KUKA KRL program: filwin67start.src

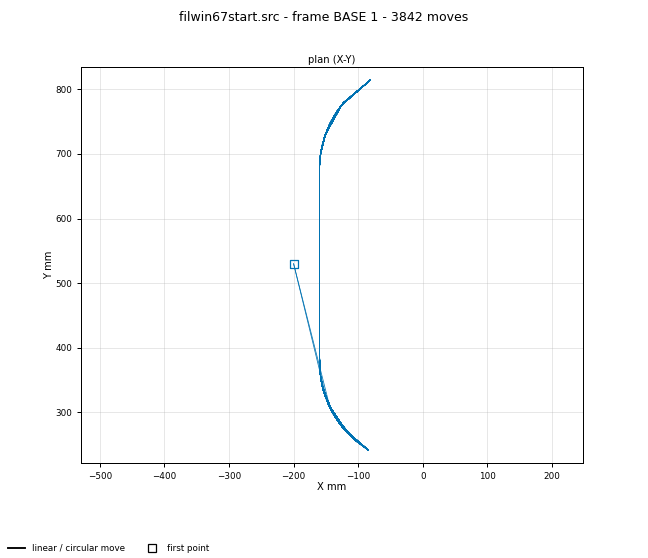
[picture p0: tool path of filwin67start.src in frame BASE 1, 3842 of 3843 moves have a stored position in this frame; points joined in program order, loops and branches not executed]
&ACCESS RVEO
&REL 11
&PARAM TEMPLATE = C:\KRC\Roboter\Template\vorgabe
&PARAM EDITMASK = *
DEF variable_helical2( )
;FOLD INI
  ;FOLD BASISTECH INI
    GLOBAL INTERRUPT DECL 3 WHEN $STOPMESS==TRUE DO IR_STOPM ( )
    INTERRUPT ON 3
    BAS (#INITMOV,0 )
  ;ENDFOLD (BASISTECH INI)
 ;FOLD USER INI


    ;Make your modifications here
  ;ENDFOLD (USER INI)
;ENDFOLD (INI)
ACTION(#AXIS_RESET,34,1000,#NOERROR,ERROR_CODE)
;FOLD PTP HOME  Vel= 100 % DEFAULT;%{PE}%MKUKATPBASIS,%CMOVE,%VPTP,%P 1:PTP, 2:HOME, 3:, 5:100, 7:DEFAULT
$BWDSTART = FALSE
PDAT_ACT=PDEFAULT
FDAT_ACT=FHOME
BAS (#PTP_PARAMS,100 )
$H_POS=XHOME
PTP  XHOME
;ENDFOLD
BAS(#TOOL,1)
BAS(#BASE,1)
$VEL_AXIS[1]=100
$VEL_AXIS[2]=100
$VEL_AXIS[3]=100
$VEL_AXIS[4]=100
$VEL_AXIS[5]=100
$VEL_AXIS[6]=100
$VEL_EXTAX[1]=100
$VEL_EXTAX[2]=100

$ACC_AXIS[1]=100
$ACC_AXIS[2]=100
$ACC_AXIS[3]=100
$ACC_AXIS[4]=100
$ACC_AXIS[5]=100
$ACC_AXIS[6]=100
$ACC_EXTAX[1]=100
$ACC_EXTAX[2]=100

;;;;;;;;; postprocessing parameters (date 2024-01-29T17:49:23.604296)
; qxconst: -159.99
; qxconstarcys: -152.5,146.5
; qE3offset: 0.00
; qyoffset: 530.00
; qswitchsplit: 3
; qthinningtol: 0.2010
;;;;;;;;;

SLIN {X  -200.000, Y  +530.000, Z    +0.000, A    +0.000, E1    +0.000, E3    +0.000, E4    +0.000}

SLIN {X  -143.479, Y  +306.716, Z    +0.000, E1   +71.847, E3  -282.582}
HALT
SPLINE
SPL {X  -140.298, Y  +300.601, Z    +0.000, E1   +71.461, E3  -275.826}
SPL {X  -137.001, Y  +294.872, Z    +0.000, E1   +71.048, E3  -269.318}
SPL {X  -133.301, Y  +289.026, Z    +0.000, E1   +70.567, E3  -262.531}
SPL {X  -129.603, Y  +283.692, Z    +0.000, E1   +70.051, E3  -256.231}
SPL {X  -125.807, Y  +278.659, Z    +0.000, E1   +69.508, E3  -250.273}
SPL {X  -122.086, Y  +274.099, Z    +0.000, E1   +68.932, E3  -244.895}
SPL {X   -84.117, Y  +241.407, Z    +0.000, E1   +58.224, E3  -154.012}
ENDSPLINE

SPLINE
SPL {X  -116.986, Y  +268.362, Z    +0.000, E1   +53.233, E3   +39.903}
SPL {X  -146.319, Y  +312.789, Z    +0.000, E1   +44.152, E3   +70.369}
SPL {X  -157.053, Y  +346.986, Z    +0.000, E1   +27.437, E3   +78.400}
SPL {X  -159.518, Y  +365.226, Z    +0.000, E1   +13.562, E3   +80.266}
SPL {X  -159.976, Y  +375.387, Z    +0.000, E1    +4.229, E3   +80.701}
SPL {X  -159.990, Y  +379.485, Z    +0.000, E1    +0.028, E3   +80.746}
SPL {X  -159.990, Y  +381.270, Z    +0.000, E1    -3.383, E3   +80.764}
SPL {X  -159.990, Y  +386.246, Z    +0.000, E1   -14.704, E3   +80.921}
SPL {X  -159.990, Y  +394.075, Z    +0.000, E1   -32.836, E3   +81.482}
SPL {X  -159.990, Y  +405.152, Z    +0.000, E1   -50.697, E3   +82.906}
SPL {X  -159.990, Y  +423.293, Z    +0.000, E1   -63.280, E3   +86.907}
SPL {X  -159.990, Y  +493.649, Z    +0.000, E1   -71.671, E3  +112.611}
SPL {X  -159.990, Y  +662.531, Z    +0.000, E1   -73.010, E3  +199.434}
SPL {X  -159.805, Y  +684.185, Z    +0.000, E1   -72.979, E3  +213.718}
SPL {X  -158.295, Y  +699.729, Z    +0.000, E1   -72.830, E3  +225.389}
SPL {X  -155.857, Y  +712.630, Z    +0.000, E1   -72.572, E3  +236.318}
SPL {X  -153.206, Y  +722.596, Z    +0.000, E1   -72.287, E3  +245.499}
SPL {X  -150.445, Y  +730.933, Z    +0.000, E1   -71.979, E3  +253.709}
SPL {X  -147.389, Y  +738.737, Z    +0.000, E1   -71.634, E3  +261.782}
SPL {X  -144.044, Y  +746.129, Z    +0.000, E1   -71.236, E3  +269.776}
SPL {X  -140.684, Y  +752.689, Z    +0.000, E1   -70.820, E3  +277.151}
SPL {X  -137.335, Y  +758.572, Z    +0.000, E1   -70.388, E3  +283.959}
SPL {X  -133.651, Y  +764.444, Z    +0.000, E1   -69.897, E3  +290.911}
SPL {X  -129.492, Y  +770.461, Z    +0.000, E1   -69.311, E3  +298.151}
SPL {X  -125.168, Y  +776.148, Z    +0.000, E1   -68.666, E3  +305.027}
SPL {X  -122.036, Y  +779.960, Z    +0.000, E1   -68.144, E3  +309.631}
SPL {X   -80.879, Y  +814.541, Z    +0.000, E1   -55.704, E3  +430.948}
ENDSPLINE

SPLINE
SPL {X  -125.518, Y  +775.707, Z    +0.000, E1   -52.189, E3  +602.426}
SPL {X  -144.748, Y  +744.653, Z    +0.000, E1   -45.208, E3  +620.621}
SPL {X  -153.147, Y  +722.791, Z    +0.000, E1   -36.417, E3  +627.017}
SPL {X  -157.402, Y  +705.160, Z    +0.000, E1   -26.108, E3  +630.112}
SPL {X  -159.480, Y  +689.270, Z    +0.000, E1   -14.023, E3  +631.678}
SPL {X  -159.986, Y  +677.650, Z    +0.000, E1    -3.291, E3  +632.172}
SPL {X  -159.990, Y  +674.500, Z    +0.000, E1    +0.000, E3  +632.203}
SPL {X  -159.990, Y  +672.716, Z    +0.000, E1    +3.405, E3  +632.219}
SPL {X  -159.990, Y  +668.521, Z    +0.000, E1   +13.007, E3  +632.338}
SPL {X  -159.990, Y  +664.286, Z    +0.000, E1   +23.338, E3  +632.570}
SPL {X  -159.990, Y  +658.431, Z    +0.000, E1   +35.998, E3  +633.065}
SPL {X  -159.990, Y  +650.524, Z    +0.000, E1   +48.779, E3  +634.053}
SPL {X  -159.990, Y  +641.022, Z    +0.000, E1   +57.726, E3  +635.920}
SPL {X  -159.990, Y  +617.987, Z    +0.000, E1   +67.134, E3  +641.815}
SPL {X  -159.990, Y  +532.407, Z    +0.000, E1   +73.084, E3  +672.722}
SPL {X  -159.990, Y  +390.607, Z    +0.000, E1   +73.632, E3  +744.258}
SPL {X  -159.886, Y  +371.742, Z    +0.000, E1   +73.650, E3  +756.045}
SPL {X  -157.928, Y  +351.899, Z    +0.000, E1   +73.451, E3  +770.479}
ENDSPLINE

SPLINE
SPL {X  -159.990, Y  +380.170, Z    +0.000, E1   +69.785, E3  +786.619}
ENDSPLINE

SPLINE
SPL {X  -158.227, Y  +353.814, Z    +0.000, E1   +70.663, E3  +798.512}
SPL {X  -155.560, Y  +340.111, Z    +0.000, E1   +70.976, E3  +805.534}
SPL {X  -151.918, Y  +327.322, Z    +0.000, E1   +71.266, E3  +811.878}
SPL {X  -144.697, Y  +309.238, Z    +0.000, E1   +71.848, E3  +818.828}
SPL {X  -140.298, Y  +300.601, Z    +0.000, E1   +71.461, E3  +827.115}
SPL {X  -137.001, Y  +294.872, Z    +0.000, E1   +71.048, E3  +833.623}
SPL {X  -133.301, Y  +289.026, Z    +0.000, E1   +70.567, E3  +840.410}
SPL {X  -129.603, Y  +283.692, Z    +0.000, E1   +70.051, E3  +846.710}
SPL {X  -125.807, Y  +278.659, Z    +0.000, E1   +69.508, E3  +852.669}
SPL {X  -122.086, Y  +274.099, Z    +0.000, E1   +68.932, E3  +858.046}
SPL {X   -84.117, Y  +241.407, Z    +0.000, E1   +58.224, E3  +948.929}
ENDSPLINE

SPLINE
SPL {X  -106.708, Y  +258.294, Z    +0.000, E1   +53.789, E3 +1127.716}
SPL {X  -137.973, Y  +296.505, Z    +0.000, E1   +48.844, E3 +1166.496}
SPL {X  -154.359, Y  +335.426, Z    +0.000, E1   +34.338, E3 +1179.392}
SPL {X  -159.279, Y  +362.429, Z    +0.000, E1   +16.013, E3 +1182.992}
SPL {X  -159.976, Y  +375.387, Z    +0.000, E1    +4.229, E3 +1183.643}
SPL {X  -159.990, Y  +379.485, Z    +0.000, E1    +0.028, E3 +1183.688}
SPL {X  -159.990, Y  +381.270, Z    +0.000, E1    -3.383, E3 +1183.705}
SPL {X  -159.990, Y  +386.246, Z    +0.000, E1   -14.704, E3 +1183.862}
SPL {X  -159.990, Y  +394.075, Z    +0.000, E1   -32.836, E3 +1184.423}
SPL {X  -159.990, Y  +405.152, Z    +0.000, E1   -50.697, E3 +1185.847}
SPL {X  -159.990, Y  +423.293, Z    +0.000, E1   -63.280, E3 +1189.849}
SPL {X  -159.990, Y  +493.649, Z    +0.000, E1   -71.671, E3 +1215.552}
SPL {X  -159.990, Y  +662.531, Z    +0.000, E1   -73.010, E3 +1302.376}
SPL {X  -159.805, Y  +684.185, Z    +0.000, E1   -72.979, E3 +1316.660}
SPL {X  -158.739, Y  +696.464, Z    +0.000, E1   -72.862, E3 +1325.778}
SPL {X  -156.417, Y  +710.124, Z    +0.000, E1   -72.650, E3 +1337.002}
SPL {X  -153.206, Y  +722.596, Z    +0.000, E1   -72.287, E3 +1348.440}
SPL {X  -150.445, Y  +730.933, Z    +0.000, E1   -71.979, E3 +1356.650}
SPL {X  -147.389, Y  +738.737, Z    +0.000, E1   -71.634, E3 +1364.723}
SPL {X  -144.044, Y  +746.129, Z    +0.000, E1   -71.236, E3 +1372.717}
SPL {X  -140.684, Y  +752.689, Z    +0.000, E1   -70.820, E3 +1380.092}
SPL {X  -137.335, Y  +758.572, Z    +0.000, E1   -70.388, E3 +1386.900}
SPL {X  -133.651, Y  +764.444, Z    +0.000, E1   -69.897, E3 +1393.852}
SPL {X  -129.492, Y  +770.461, Z    +0.000, E1   -69.311, E3 +1401.092}
SPL {X  -125.168, Y  +776.148, Z    +0.000, E1   -68.666, E3 +1407.968}
SPL {X  -122.036, Y  +779.960, Z    +0.000, E1   -68.144, E3 +1412.572}
SPL {X   -80.879, Y  +814.541, Z    +0.000, E1   -55.704, E3 +1533.889}
ENDSPLINE

SPLINE
SPL {X  -125.518, Y  +775.707, Z    +0.000, E1   -52.189, E3 +1705.367}
SPL {X  -144.748, Y  +744.653, Z    +0.000, E1   -45.208, E3 +1723.563}
SPL {X  -153.147, Y  +722.791, Z    +0.000, E1   -36.417, E3 +1729.958}
SPL {X  -157.402, Y  +705.160, Z    +0.000, E1   -26.108, E3 +1733.054}
SPL {X  -159.480, Y  +689.270, Z    +0.000, E1   -14.023, E3 +1734.619}
SPL {X  -159.986, Y  +677.650, Z    +0.000, E1    -3.291, E3 +1735.114}
SPL {X  -159.990, Y  +674.500, Z    +0.000, E1    +0.000, E3 +1735.144}
SPL {X  -159.990, Y  +672.716, Z    +0.000, E1    +3.405, E3 +1735.161}
SPL {X  -159.990, Y  +668.521, Z    +0.000, E1   +13.007, E3 +1735.280}
SPL {X  -159.990, Y  +664.286, Z    +0.000, E1   +23.338, E3 +1735.511}
SPL {X  -159.990, Y  +658.431, Z    +0.000, E1   +35.998, E3 +1736.006}
SPL {X  -159.990, Y  +650.524, Z    +0.000, E1   +48.779, E3 +1736.994}
SPL {X  -159.990, Y  +641.022, Z    +0.000, E1   +57.726, E3 +1738.861}
SPL {X  -159.990, Y  +617.987, Z    +0.000, E1   +67.134, E3 +1744.757}
SPL {X  -159.990, Y  +532.407, Z    +0.000, E1   +73.084, E3 +1775.663}
SPL {X  -159.990, Y  +382.957, Z    +0.000, E1   +73.647, E3 +1851.923}
SPL {X  -159.615, Y  +366.548, Z    +0.000, E1   +73.602, E3 +1862.565}
SPL {X  -157.928, Y  +351.899, Z    +0.000, E1   +73.451, E3 +1873.420}
ENDSPLINE

SPLINE
SPL {X  -159.990, Y  +387.996, Z    +0.000, E1   +69.509, E3 +1885.850}
ENDSPLINE

SPLINE
SPL {X  -159.889, Y  +371.819, Z    +0.000, E1   +70.046, E3 +1893.577}
SPL {X  -158.227, Y  +353.814, Z    +0.000, E1   +70.663, E3 +1901.454}
SPL {X  -154.257, Y  +335.055, Z    +0.000, E1   +71.089, E3 +1911.082}
SPL {X  -148.153, Y  +317.104, Z    +0.000, E1   +71.658, E3 +1918.227}
SPL {X  -143.479, Y  +306.716, Z    +0.000, E1   +71.847, E3 +1923.301}
SPL {X  -140.298, Y  +300.601, Z    +0.000, E1   +71.461, E3 +1930.056}
SPL {X  -135.903, Y  +293.078, Z    +0.000, E1   +70.930, E3 +1938.594}
SPL {X  -130.487, Y  +284.926, Z    +0.000, E1   +70.202, E3 +1948.153}
SPL {X  -125.807, Y  +278.659, Z    +0.000, E1   +69.508, E3 +1955.610}
SPL {X  -122.967, Y  +275.148, Z    +0.000, E1   +69.053, E3 +1959.779}
SPL {X  -121.236, Y  +273.103, Z    +0.000, E1   +68.779, E3 +1962.164}
SPL {X   -84.117, Y  +241.407, Z    +0.000, E1   +58.224, E3 +2051.870}
ENDSPLINE

SPLINE
SPL {X  -116.986, Y  +268.362, Z    +0.000, E1   +53.233, E3 +2245.785}
SPL {X  -146.319, Y  +312.789, Z    +0.000, E1   +44.152, E3 +2276.252}
SPL {X  -157.053, Y  +346.986, Z    +0.000, E1   +27.437, E3 +2284.283}
SPL {X  -159.518, Y  +365.226, Z    +0.000, E1   +13.562, E3 +2286.148}
SPL {X  -159.976, Y  +375.387, Z    +0.000, E1    +4.229, E3 +2286.584}
SPL {X  -159.990, Y  +379.485, Z    +0.000, E1    +0.028, E3 +2286.629}
SPL {X  -159.990, Y  +381.270, Z    +0.000, E1    -3.383, E3 +2286.646}
SPL {X  -159.990, Y  +386.246, Z    +0.000, E1   -14.704, E3 +2286.803}
SPL {X  -159.990, Y  +394.075, Z    +0.000, E1   -32.836, E3 +2287.364}
SPL {X  -159.990, Y  +405.152, Z    +0.000, E1   -50.697, E3 +2288.788}
SPL {X  -159.990, Y  +423.293, Z    +0.000, E1   -63.280, E3 +2292.790}
SPL {X  -159.990, Y  +493.649, Z    +0.000, E1   -71.671, E3 +2318.494}
SPL {X  -159.990, Y  +662.531, Z    +0.000, E1   -73.010, E3 +2405.317}
SPL {X  -159.805, Y  +684.185, Z    +0.000, E1   -72.979, E3 +2419.601}
SPL {X  -158.295, Y  +699.729, Z    +0.000, E1   -72.830, E3 +2431.271}
SPL {X  -155.857, Y  +712.630, Z    +0.000, E1   -72.572, E3 +2442.200}
SPL {X  -153.206, Y  +722.596, Z    +0.000, E1   -72.287, E3 +2451.381}
SPL {X  -150.445, Y  +730.933, Z    +0.000, E1   -71.979, E3 +2459.591}
SPL {X  -147.389, Y  +738.737, Z    +0.000, E1   -71.634, E3 +2467.664}
SPL {X  -144.044, Y  +746.129, Z    +0.000, E1   -71.236, E3 +2475.658}
SPL {X  -140.684, Y  +752.689, Z    +0.000, E1   -70.820, E3 +2483.034}
SPL {X  -136.099, Y  +760.606, Z    +0.000, E1   -70.253, E3 +2492.189}
SPL {X  -131.456, Y  +767.693, Z    +0.000, E1   -69.587, E3 +2500.701}
SPL {X  -127.440, Y  +773.226, Z    +0.000, E1   -69.006, E3 +2507.385}
SPL {X  -123.127, Y  +778.659, Z    +0.000, E1   -68.349, E3 +2513.927}
SPL {X   -80.879, Y  +814.541, Z    +0.000, E1   -55.704, E3 +2636.831}
ENDSPLINE

SPLINE
SPL {X  -125.518, Y  +775.707, Z    +0.000, E1   -52.189, E3 +2808.308}
SPL {X  -150.797, Y  +729.951, Z    +0.000, E1   -39.777, E3 +2831.043}
SPL {X  -158.456, Y  +698.602, Z    +0.000, E1   -21.523, E3 +2836.746}
SPL {X  -159.738, Y  +685.469, Z    +0.000, E1   -10.595, E3 +2837.800}
SPL {X  -159.986, Y  +677.650, Z    +0.000, E1    -3.291, E3 +2838.055}
SPL {X  -159.990, Y  +674.500, Z    +0.000, E1    +0.000, E3 +2838.085}
SPL {X  -159.990, Y  +672.716, Z    +0.000, E1    +3.405, E3 +2838.102}
SPL {X  -159.990, Y  +668.521, Z    +0.000, E1   +13.007, E3 +2838.221}
SPL {X  -159.990, Y  +662.839, Z    +0.000, E1   +26.519, E3 +2838.563}
SPL {X  -159.990, Y  +653.836, Z    +0.000, E1   +43.967, E3 +2839.493}
SPL {X  -159.990, Y  +641.022, Z    +0.000, E1   +57.726, E3 +2841.802}
SPL {X  -159.990, Y  +617.987, Z    +0.000, E1   +67.134, E3 +2847.698}
SPL {X  -159.990, Y  +532.407, Z    +0.000, E1   +73.084, E3 +2878.605}
SPL {X  -159.990, Y  +382.957, Z    +0.000, E1   +73.647, E3 +2954.864}
SPL {X  -159.615, Y  +366.548, Z    +0.000, E1   +73.602, E3 +2965.507}
SPL {X  -157.928, Y  +351.899, Z    +0.000, E1   +73.451, E3 +2976.361}
ENDSPLINE

SPLINE
SPL {X  -159.990, Y  +380.170, Z    +0.000, E1   +69.785, E3 +2992.501}
ENDSPLINE

SPLINE
SPL {X  -158.227, Y  +353.814, Z    +0.000, E1   +70.663, E3 +3004.395}
SPL {X  -154.257, Y  +335.055, Z    +0.000, E1   +71.089, E3 +3014.023}
SPL {X  -148.153, Y  +317.104, Z    +0.000, E1   +71.658, E3 +3021.168}
SPL {X  -143.479, Y  +306.716, Z    +0.000, E1   +71.847, E3 +3026.242}
SPL {X  -140.298, Y  +300.601, Z    +0.000, E1   +71.461, E3 +3032.997}
SPL {X  -137.001, Y  +294.872, Z    +0.000, E1   +71.048, E3 +3039.506}
SPL {X  -133.301, Y  +289.026, Z    +0.000, E1   +70.567, E3 +3046.292}
SPL {X  -128.648, Y  +282.387, Z    +0.000, E1   +69.939, E3 +3054.107}
SPL {X  -125.063, Y  +277.720, Z    +0.000, E1   +69.378, E3 +3059.683}
SPL {X  -122.086, Y  +274.099, Z    +0.000, E1   +68.932, E3 +3063.928}
SPL {X   -84.117, Y  +241.407, Z    +0.000, E1   +58.224, E3 +3154.811}
ENDSPLINE

SPLINE
SPL {X  -106.708, Y  +258.294, Z    +0.000, E1   +53.789, E3 +3333.598}
SPL {X  -137.973, Y  +296.505, Z    +0.000, E1   +48.844, E3 +3372.378}
SPL {X  -154.359, Y  +335.426, Z    +0.000, E1   +34.338, E3 +3385.274}
SPL {X  -159.279, Y  +362.429, Z    +0.000, E1   +16.013, E3 +3388.874}
SPL {X  -159.976, Y  +375.387, Z    +0.000, E1    +4.229, E3 +3389.525}
SPL {X  -159.990, Y  +379.485, Z    +0.000, E1    +0.028, E3 +3389.570}
SPL {X  -159.990, Y  +381.270, Z    +0.000, E1    -3.383, E3 +3389.587}
SPL {X  -159.990, Y  +386.246, Z    +0.000, E1   -14.704, E3 +3389.745}
SPL {X  -159.990, Y  +394.075, Z    +0.000, E1   -32.836, E3 +3390.305}
SPL {X  -159.990, Y  +405.152, Z    +0.000, E1   -50.697, E3 +3391.730}
SPL {X  -159.990, Y  +423.293, Z    +0.000, E1   -63.280, E3 +3395.731}
SPL {X  -159.990, Y  +493.649, Z    +0.000, E1   -71.671, E3 +3421.435}
SPL {X  -159.990, Y  +662.531, Z    +0.000, E1   -73.010, E3 +3508.258}
SPL {X  -159.805, Y  +684.185, Z    +0.000, E1   -72.979, E3 +3522.542}
SPL {X  -158.739, Y  +696.464, Z    +0.000, E1   -72.862, E3 +3531.661}
SPL {X  -156.417, Y  +710.124, Z    +0.000, E1   -72.650, E3 +3542.884}
SPL {X  -153.206, Y  +722.596, Z    +0.000, E1   -72.287, E3 +3554.322}
SPL {X  -150.445, Y  +730.933, Z    +0.000, E1   -71.979, E3 +3562.532}
SPL {X  -147.389, Y  +738.737, Z    +0.000, E1   -71.634, E3 +3570.605}
SPL {X  -144.044, Y  +746.129, Z    +0.000, E1   -71.236, E3 +3578.600}
SPL {X  -140.684, Y  +752.689, Z    +0.000, E1   -70.820, E3 +3585.975}
SPL {X  -137.335, Y  +758.572, Z    +0.000, E1   -70.388, E3 +3592.782}
SPL {X  -133.651, Y  +764.444, Z    +0.000, E1   -69.897, E3 +3599.734}
SPL {X  -130.650, Y  +768.844, Z    +0.000, E1   -69.455, E3 +3605.055}
SPL {X  -127.440, Y  +773.226, Z    +0.000, E1   -69.006, E3 +3610.326}
SPL {X  -123.127, Y  +778.659, Z    +0.000, E1   -68.349, E3 +3616.868}
SPL {X   -80.879, Y  +814.541, Z    +0.000, E1   -55.704, E3 +3739.772}
ENDSPLINE

SPLINE
SPL {X  -125.518, Y  +775.707, Z    +0.000, E1   -52.189, E3 +3911.249}
SPL {X  -144.748, Y  +744.653, Z    +0.000, E1   -45.208, E3 +3929.445}
SPL {X  -153.147, Y  +722.791, Z    +0.000, E1   -36.417, E3 +3935.841}
SPL {X  -157.402, Y  +705.160, Z    +0.000, E1   -26.108, E3 +3938.936}
SPL {X  -159.480, Y  +689.270, Z    +0.000, E1   -14.023, E3 +3940.502}
SPL {X  -159.986, Y  +677.650, Z    +0.000, E1    -3.291, E3 +3940.996}
SPL {X  -159.990, Y  +674.500, Z    +0.000, E1    +0.000, E3 +3941.026}
SPL {X  -159.990, Y  +672.716, Z    +0.000, E1    +3.405, E3 +3941.043}
SPL {X  -159.990, Y  +668.521, Z    +0.000, E1   +13.007, E3 +3941.162}
SPL {X  -159.990, Y  +664.286, Z    +0.000, E1   +23.338, E3 +3941.393}
SPL {X  -159.990, Y  +658.431, Z    +0.000, E1   +35.998, E3 +3941.888}
SPL {X  -159.990, Y  +650.524, Z    +0.000, E1   +48.779, E3 +3942.877}
SPL {X  -159.990, Y  +641.022, Z    +0.000, E1   +57.726, E3 +3944.743}
SPL {X  -159.990, Y  +617.987, Z    +0.000, E1   +67.134, E3 +3950.639}
SPL {X  -159.990, Y  +532.407, Z    +0.000, E1   +73.084, E3 +3981.546}
SPL {X  -159.990, Y  +382.957, Z    +0.000, E1   +73.647, E3 +4057.805}
SPL {X  -159.615, Y  +366.548, Z    +0.000, E1   +73.602, E3 +4068.448}
SPL {X  -157.928, Y  +351.899, Z    +0.000, E1   +73.451, E3 +4079.302}
ENDSPLINE

SPLINE
SPL {X  -159.990, Y  +387.996, Z    +0.000, E1   +69.509, E3 +4091.732}
ENDSPLINE

SPLINE
SPL {X  -159.889, Y  +371.819, Z    +0.000, E1   +70.046, E3 +4099.459}
SPL {X  -158.227, Y  +353.814, Z    +0.000, E1   +70.663, E3 +4107.336}
SPL {X  -154.257, Y  +335.055, Z    +0.000, E1   +71.089, E3 +4116.964}
SPL {X  -148.153, Y  +317.104, Z    +0.000, E1   +71.658, E3 +4124.109}
SPL {X  -143.479, Y  +306.716, Z    +0.000, E1   +71.847, E3 +4129.183}
SPL {X  -140.298, Y  +300.601, Z    +0.000, E1   +71.461, E3 +4135.939}
SPL {X  -135.903, Y  +293.078, Z    +0.000, E1   +70.930, E3 +4144.476}
SPL {X  -130.487, Y  +284.926, Z    +0.000, E1   +70.202, E3 +4154.036}
SPL {X  -125.807, Y  +278.659, Z    +0.000, E1   +69.508, E3 +4161.492}
SPL {X  -122.967, Y  +275.148, Z    +0.000, E1   +69.053, E3 +4165.661}
SPL {X  -121.236, Y  +273.103, Z    +0.000, E1   +68.779, E3 +4168.046}
SPL {X   -84.117, Y  +241.407, Z    +0.000, E1   +58.224, E3 +4257.752}
ENDSPLINE

SPLINE
SPL {X  -116.986, Y  +268.362, Z    +0.000, E1   +53.233, E3 +4451.668}
SPL {X  -146.319, Y  +312.789, Z    +0.000, E1   +44.152, E3 +4482.134}
SPL {X  -157.053, Y  +346.986, Z    +0.000, E1   +27.437, E3 +4490.165}
SPL {X  -159.518, Y  +365.226, Z    +0.000, E1   +13.562, E3 +4492.031}
SPL {X  -159.976, Y  +375.387, Z    +0.000, E1    +4.229, E3 +4492.466}
SPL {X  -159.990, Y  +379.485, Z    +0.000, E1    +0.028, E3 +4492.511}
SPL {X  -159.990, Y  +381.270, Z    +0.000, E1    -3.383, E3 +4492.528}
SPL {X  -159.990, Y  +386.246, Z    +0.000, E1   -14.704, E3 +4492.686}
SPL {X  -159.990, Y  +394.075, Z    +0.000, E1   -32.836, E3 +4493.246}
SPL {X  -159.990, Y  +405.152, Z    +0.000, E1   -50.697, E3 +4494.671}
SPL {X  -159.990, Y  +423.293, Z    +0.000, E1   -63.280, E3 +4498.672}
SPL {X  -159.990, Y  +493.649, Z    +0.000, E1   -71.671, E3 +4524.376}
SPL {X  -159.990, Y  +662.531, Z    +0.000, E1   -73.010, E3 +4611.199}
SPL {X  -159.805, Y  +684.185, Z    +0.000, E1   -72.979, E3 +4625.483}
SPL {X  -158.295, Y  +699.729, Z    +0.000, E1   -72.830, E3 +4637.153}
SPL {X  -155.857, Y  +712.630, Z    +0.000, E1   -72.572, E3 +4648.082}
SPL {X  -153.206, Y  +722.596, Z    +0.000, E1   -72.287, E3 +4657.263}
SPL {X  -150.445, Y  +730.933, Z    +0.000, E1   -71.979, E3 +4665.474}
SPL {X  -147.389, Y  +738.737, Z    +0.000, E1   -71.634, E3 +4673.546}
SPL {X  -144.044, Y  +746.129, Z    +0.000, E1   -71.236, E3 +4681.541}
SPL {X  -140.684, Y  +752.689, Z    +0.000, E1   -70.820, E3 +4688.916}
SPL {X  -136.099, Y  +760.606, Z    +0.000, E1   -70.253, E3 +4698.071}
SPL {X  -131.456, Y  +767.693, Z    +0.000, E1   -69.587, E3 +4706.583}
SPL {X  -127.440, Y  +773.226, Z    +0.000, E1   -69.006, E3 +4713.267}
SPL {X  -123.127, Y  +778.659, Z    +0.000, E1   -68.349, E3 +4719.809}
SPL {X   -80.879, Y  +814.541, Z    +0.000, E1   -55.704, E3 +4842.713}
ENDSPLINE

SPLINE
SPL {X  -125.518, Y  +775.707, Z    +0.000, E1   -52.189, E3 +5014.190}
SPL {X  -144.748, Y  +744.653, Z    +0.000, E1   -45.208, E3 +5032.386}
SPL {X  -153.147, Y  +722.791, Z    +0.000, E1   -36.417, E3 +5038.782}
SPL {X  -158.456, Y  +698.602, Z    +0.000, E1   -21.523, E3 +5042.628}
SPL {X  -159.738, Y  +685.469, Z    +0.000, E1   -10.595, E3 +5043.682}
SPL {X  -159.986, Y  +677.650, Z    +0.000, E1    -3.291, E3 +5043.937}
SPL {X  -159.990, Y  +674.500, Z    +0.000, E1    +0.000, E3 +5043.968}
SPL {X  -159.990, Y  +672.716, Z    +0.000, E1    +3.405, E3 +5043.984}
SPL {X  -159.990, Y  +668.521, Z    +0.000, E1   +13.007, E3 +5044.103}
SPL {X  -159.990, Y  +664.286, Z    +0.000, E1   +23.338, E3 +5044.335}
SPL {X  -159.990, Y  +658.431, Z    +0.000, E1   +35.998, E3 +5044.829}
SPL {X  -159.990, Y  +650.524, Z    +0.000, E1   +48.779, E3 +5045.818}
SPL {X  -159.990, Y  +641.022, Z    +0.000, E1   +57.726, E3 +5047.685}
SPL {X  -159.990, Y  +617.987, Z    +0.000, E1   +67.134, E3 +5053.580}
SPL {X  -159.990, Y  +532.407, Z    +0.000, E1   +73.084, E3 +5084.487}
SPL {X  -159.990, Y  +390.607, Z    +0.000, E1   +73.632, E3 +5156.023}
SPL {X  -159.886, Y  +371.742, Z    +0.000, E1   +73.650, E3 +5167.810}
SPL {X  -157.928, Y  +351.899, Z    +0.000, E1   +73.451, E3 +5182.243}
ENDSPLINE

SPLINE
SPL {X  -159.990, Y  +380.170, Z    +0.000, E1   +69.785, E3 +5198.384}
ENDSPLINE

SPLINE
SPL {X  -158.227, Y  +353.814, Z    +0.000, E1   +70.663, E3 +5210.277}
SPL {X  -154.257, Y  +335.055, Z    +0.000, E1   +71.089, E3 +5219.905}
SPL {X  -148.153, Y  +317.104, Z    +0.000, E1   +71.658, E3 +5227.051}
SPL {X  -143.479, Y  +306.716, Z    +0.000, E1   +71.847, E3 +5232.124}
SPL {X  -140.298, Y  +300.601, Z    +0.000, E1   +71.461, E3 +5238.880}
SPL {X  -137.001, Y  +294.872, Z    +0.000, E1   +71.048, E3 +5245.388}
SPL {X  -133.301, Y  +289.026, Z    +0.000, E1   +70.567, E3 +5252.175}
SPL {X  -128.648, Y  +282.387, Z    +0.000, E1   +69.939, E3 +5259.990}
SPL {X  -125.063, Y  +277.720, Z    +0.000, E1   +69.378, E3 +5265.565}
SPL {X  -122.086, Y  +274.099, Z    +0.000, E1   +68.932, E3 +5269.811}
SPL {X   -84.117, Y  +241.407, Z    +0.000, E1   +58.224, E3 +5360.693}
ENDSPLINE

SPLINE
SPL {X  -106.708, Y  +258.294, Z    +0.000, E1   +53.789, E3 +5539.480}
SPL {X  -137.973, Y  +296.505, Z    +0.000, E1   +48.844, E3 +5578.261}
SPL {X  -154.359, Y  +335.426, Z    +0.000, E1   +34.338, E3 +5591.157}
SPL {X  -159.279, Y  +362.429, Z    +0.000, E1   +16.013, E3 +5594.757}
SPL {X  -159.976, Y  +375.387, Z    +0.000, E1    +4.229, E3 +5595.407}
SPL {X  -159.990, Y  +379.485, Z    +0.000, E1    +0.028, E3 +5595.452}
SPL {X  -159.990, Y  +381.270, Z    +0.000, E1    -3.383, E3 +5595.469}
SPL {X  -159.990, Y  +386.246, Z    +0.000, E1   -14.704, E3 +5595.627}
SPL {X  -159.990, Y  +394.075, Z    +0.000, E1   -32.836, E3 +5596.188}
SPL {X  -159.990, Y  +405.152, Z    +0.000, E1   -50.697, E3 +5597.612}
SPL {X  -159.990, Y  +423.293, Z    +0.000, E1   -63.280, E3 +5601.613}
SPL {X  -159.990, Y  +493.649, Z    +0.000, E1   -71.671, E3 +5627.317}
SPL {X  -159.990, Y  +662.531, Z    +0.000, E1   -73.010, E3 +5714.140}
SPL {X  -159.805, Y  +684.185, Z    +0.000, E1   -72.979, E3 +5728.424}
SPL {X  -158.739, Y  +696.464, Z    +0.000, E1   -72.862, E3 +5737.543}
SPL {X  -156.417, Y  +710.124, Z    +0.000, E1   -72.650, E3 +5748.766}
SPL {X  -153.206, Y  +722.596, Z    +0.000, E1   -72.287, E3 +5760.204}
SPL {X  -150.445, Y  +730.933, Z    +0.000, E1   -71.979, E3 +5768.415}
SPL {X  -147.389, Y  +738.737, Z    +0.000, E1   -71.634, E3 +5776.487}
SPL {X  -144.044, Y  +746.129, Z    +0.000, E1   -71.236, E3 +5784.482}
SPL {X  -140.684, Y  +752.689, Z    +0.000, E1   -70.820, E3 +5791.857}
SPL {X  -137.335, Y  +758.572, Z    +0.000, E1   -70.388, E3 +5798.664}
SPL {X  -133.651, Y  +764.444, Z    +0.000, E1   -69.897, E3 +5805.617}
SPL {X  -130.650, Y  +768.844, Z    +0.000, E1   -69.455, E3 +5810.938}
SPL {X  -127.440, Y  +773.226, Z    +0.000, E1   -69.006, E3 +5816.208}
SPL {X  -123.127, Y  +778.659, Z    +0.000, E1   -68.349, E3 +5822.750}
SPL {X   -80.879, Y  +814.541, Z    +0.000, E1   -55.704, E3 +5945.654}
ENDSPLINE

SPLINE
SPL {X  -125.518, Y  +775.707, Z    +0.000, E1   -52.189, E3 +6117.132}
SPL {X  -150.797, Y  +729.951, Z    +0.000, E1   -39.777, E3 +6139.866}
SPL {X  -158.456, Y  +698.602, Z    +0.000, E1   -21.523, E3 +6145.569}
SPL {X  -159.738, Y  +685.469, Z    +0.000, E1   -10.595, E3 +6146.623}
SPL {X  -159.986, Y  +677.650, Z    +0.000, E1    -3.291, E3 +6146.878}
SPL {X  -159.990, Y  +674.500, Z    +0.000, E1    +0.000, E3 +6146.909}
SPL {X  -159.990, Y  +672.716, Z    +0.000, E1    +3.405, E3 +6146.925}
SPL {X  -159.990, Y  +668.521, Z    +0.000, E1   +13.007, E3 +6147.044}
SPL {X  -159.990, Y  +662.839, Z    +0.000, E1   +26.519, E3 +6147.387}
SPL {X  -159.990, Y  +653.836, Z    +0.000, E1   +43.967, E3 +6148.317}
SPL {X  -159.990, Y  +641.022, Z    +0.000, E1   +57.726, E3 +6150.626}
SPL {X  -159.990, Y  +617.987, Z    +0.000, E1   +67.134, E3 +6156.521}
SPL {X  -159.990, Y  +532.407, Z    +0.000, E1   +73.084, E3 +6187.428}
SPL {X  -159.990, Y  +382.957, Z    +0.000, E1   +73.647, E3 +6263.688}
SPL {X  -159.615, Y  +366.548, Z    +0.000, E1   +73.602, E3 +6274.330}
SPL {X  -157.928, Y  +351.899, Z    +0.000, E1   +73.451, E3 +6285.184}
ENDSPLINE

SPLINE
SPL {X  -159.990, Y  +380.170, Z    +0.000, E1   +69.785, E3 +6301.325}
ENDSPLINE

SPLINE
SPL {X  -158.227, Y  +353.814, Z    +0.000, E1   +70.663, E3 +6313.218}
SPL {X  -154.257, Y  +335.055, Z    +0.000, E1   +71.089, E3 +6322.846}
SPL {X  -148.153, Y  +317.104, Z    +0.000, E1   +71.658, E3 +6329.992}
SPL {X  -143.479, Y  +306.716, Z    +0.000, E1   +71.847, E3 +6335.065}
SPL {X  -140.298, Y  +300.601, Z    +0.000, E1   +71.461, E3 +6341.821}
SPL {X  -137.001, Y  +294.872, Z    +0.000, E1   +71.048, E3 +6348.329}
SPL {X  -133.301, Y  +289.026, Z    +0.000, E1   +70.567, E3 +6355.116}
SPL {X  -129.603, Y  +283.692, Z    +0.000, E1   +70.051, E3 +6361.416}
SPL {X  -125.807, Y  +278.659, Z    +0.000, E1   +69.508, E3 +6367.374}
SPL {X  -122.086, Y  +274.099, Z    +0.000, E1   +68.932, E3 +6372.752}
SPL {X   -84.117, Y  +241.407, Z    +0.000, E1   +58.224, E3 +6463.635}
ENDSPLINE

SPLINE
SPL {X  -116.986, Y  +268.362, Z    +0.000, E1   +53.233, E3 +6657.550}
SPL {X  -146.319, Y  +312.789, Z    +0.000, E1   +44.152, E3 +6688.016}
SPL {X  -157.053, Y  +346.986, Z    +0.000, E1   +27.437, E3 +6696.047}
SPL {X  -159.518, Y  +365.226, Z    +0.000, E1   +13.562, E3 +6697.913}
SPL {X  -159.976, Y  +375.387, Z    +0.000, E1    +4.229, E3 +6698.348}
SPL {X  -159.990, Y  +379.485, Z    +0.000, E1    +0.028, E3 +6698.394}
SPL {X  -159.990, Y  +381.270, Z    +0.000, E1    -3.383, E3 +6698.411}
SPL {X  -159.990, Y  +384.811, Z    +0.000, E1   -11.531, E3 +6698.501}
SPL {X  -159.990, Y  +390.180, Z    +0.000, E1   -24.142, E3 +6698.804}
SPL {X  -159.990, Y  +397.074, Z    +0.000, E1   -39.012, E3 +6699.414}
SPL {X  -159.990, Y  +405.152, Z    +0.000, E1   -50.697, E3 +6700.553}
SPL {X  -159.990, Y  +423.293, Z    +0.000, E1   -63.280, E3 +6704.554}
SPL {X  -159.990, Y  +493.649, Z    +0.000, E1   -71.671, E3 +6730.258}
SPL {X  -159.990, Y  +662.531, Z    +0.000, E1   -73.010, E3 +6817.081}
SPL {X  -159.805, Y  +684.185, Z    +0.000, E1   -72.979, E3 +6831.365}
SPL {X  -158.739, Y  +696.464, Z    +0.000, E1   -72.862, E3 +6840.484}
SPL {X  -156.417, Y  +710.124, Z    +0.000, E1   -72.650, E3 +6851.707}
SPL {X  -153.206, Y  +722.596, Z    +0.000, E1   -72.287, E3 +6863.146}
SPL {X  -150.445, Y  +730.933, Z    +0.000, E1   -71.979, E3 +6871.356}
SPL {X  -147.389, Y  +738.737, Z    +0.000, E1   -71.634, E3 +6879.429}
SPL {X  -144.044, Y  +746.129, Z    +0.000, E1   -71.236, E3 +6887.423}
SPL {X  -140.684, Y  +752.689, Z    +0.000, E1   -70.820, E3 +6894.798}
SPL {X  -137.335, Y  +758.572, Z    +0.000, E1   -70.388, E3 +6901.606}
SPL {X  -134.566, Y  +763.037, Z    +0.000, E1   -70.007, E3 +6906.902}
SPL {X  -131.456, Y  +767.693, Z    +0.000, E1   -69.587, E3 +6912.465}
SPL {X  -127.440, Y  +773.226, Z    +0.000, E1   -69.006, E3 +6919.149}
SPL {X  -123.127, Y  +778.659, Z    +0.000, E1   -68.349, E3 +6925.691}
SPL {X   -80.879, Y  +814.541, Z    +0.000, E1   -55.704, E3 +7048.595}
ENDSPLINE

SPLINE
SPL {X  -125.518, Y  +775.707, Z    +0.000, E1   -52.189, E3 +7220.073}
SPL {X  -144.748, Y  +744.653, Z    +0.000, E1   -45.208, E3 +7238.269}
SPL {X  -153.147, Y  +722.791, Z    +0.000, E1   -36.417, E3 +7244.664}
SPL {X  -157.402, Y  +705.160, Z    +0.000, E1   -26.108, E3 +7247.759}
SPL {X  -159.480, Y  +689.270, Z    +0.000, E1   -14.023, E3 +7249.325}
SPL {X  -159.986, Y  +677.650, Z    +0.000, E1    -3.291, E3 +7249.819}
SPL {X  -159.990, Y  +674.500, Z    +0.000, E1    +0.000, E3 +7249.850}
SPL {X  -159.990, Y  +672.716, Z    +0.000, E1    +3.405, E3 +7249.866}
SPL {X  -159.990, Y  +668.521, Z    +0.000, E1   +13.007, E3 +7249.985}
SPL {X  -159.990, Y  +662.839, Z    +0.000, E1   +26.519, E3 +7250.328}
SPL {X  -159.990, Y  +653.836, Z    +0.000, E1   +43.967, E3 +7251.258}
SPL {X  -159.990, Y  +641.022, Z    +0.000, E1   +57.726, E3 +7253.567}
SPL {X  -159.990, Y  +617.987, Z    +0.000, E1   +67.134, E3 +7259.463}
SPL {X  -159.990, Y  +532.407, Z    +0.000, E1   +73.084, E3 +7290.369}
SPL {X  -159.990, Y  +382.957, Z    +0.000, E1   +73.647, E3 +7366.629}
SPL {X  -159.615, Y  +366.548, Z    +0.000, E1   +73.602, E3 +7377.271}
SPL {X  -157.928, Y  +351.899, Z    +0.000, E1   +73.451, E3 +7388.126}
ENDSPLINE

SPLINE
SPL {X  -159.990, Y  +380.170, Z    +0.000, E1   +69.785, E3 +7404.266}
ENDSPLINE

SPLINE
SPL {X  -158.227, Y  +353.814, Z    +0.000, E1   +70.663, E3 +7416.159}
SPL {X  -155.560, Y  +340.111, Z    +0.000, E1   +70.976, E3 +7423.181}
SPL {X  -151.918, Y  +327.322, Z    +0.000, E1   +71.266, E3 +7429.525}
SPL {X  -144.697, Y  +309.238, Z    +0.000, E1   +71.848, E3 +7436.475}
SPL {X  -140.298, Y  +300.601, Z    +0.000, E1   +71.461, E3 +7444.762}
SPL {X  -137.001, Y  +294.872, Z    +0.000, E1   +71.048, E3 +7451.270}
SPL {X  -133.301, Y  +289.026, Z    +0.000, E1   +70.567, E3 +7458.057}
SPL {X  -129.603, Y  +283.692, Z    +0.000, E1   +70.051, E3 +7464.357}
SPL {X  -125.807, Y  +278.659, Z    +0.000, E1   +69.508, E3 +7470.316}
SPL {X  -122.086, Y  +274.099, Z    +0.000, E1   +68.932, E3 +7475.693}
SPL {X   -84.117, Y  +241.407, Z    +0.000, E1   +58.224, E3 +7566.576}
ENDSPLINE

SPLINE
SPL {X  -106.708, Y  +258.294, Z    +0.000, E1   +53.789, E3 +7745.363}
SPL {X  -137.973, Y  +296.505, Z    +0.000, E1   +48.844, E3 +7784.143}
SPL {X  -154.359, Y  +335.426, Z    +0.000, E1   +34.338, E3 +7797.039}
SPL {X  -159.279, Y  +362.429, Z    +0.000, E1   +16.013, E3 +7800.639}
SPL {X  -159.976, Y  +375.387, Z    +0.000, E1    +4.229, E3 +7801.290}
SPL {X  -159.990, Y  +379.485, Z    +0.000, E1    +0.028, E3 +7801.335}
SPL {X  -159.990, Y  +381.270, Z    +0.000, E1    -3.383, E3 +7801.352}
SPL {X  -159.990, Y  +386.246, Z    +0.000, E1   -14.704, E3 +7801.509}
SPL {X  -159.990, Y  +394.075, Z    +0.000, E1   -32.836, E3 +7802.070}
SPL {X  -159.990, Y  +405.152, Z    +0.000, E1   -50.697, E3 +7803.494}
SPL {X  -159.990, Y  +423.293, Z    +0.000, E1   -63.280, E3 +7807.496}
SPL {X  -159.990, Y  +493.649, Z    +0.000, E1   -71.671, E3 +7833.199}
SPL {X  -159.990, Y  +662.531, Z    +0.000, E1   -73.010, E3 +7920.023}
SPL {X  -159.805, Y  +684.185, Z    +0.000, E1   -72.979, E3 +7934.307}
SPL {X  -158.739, Y  +696.464, Z    +0.000, E1   -72.862, E3 +7943.425}
SPL {X  -156.417, Y  +710.124, Z    +0.000, E1   -72.650, E3 +7954.649}
SPL {X  -153.206, Y  +722.596, Z    +0.000, E1   -72.287, E3 +7966.087}
SPL {X  -150.445, Y  +730.933, Z    +0.000, E1   -71.979, E3 +7974.297}
SPL {X  -147.389, Y  +738.737, Z    +0.000, E1   -71.634, E3 +7982.370}
SPL {X  -144.044, Y  +746.129, Z    +0.000, E1   -71.236, E3 +7990.364}
SPL {X  -140.684, Y  +752.689, Z    +0.000, E1   -70.820, E3 +7997.740}
SPL {X  -137.335, Y  +758.572, Z    +0.000, E1   -70.388, E3 +8004.547}
SPL {X  -133.651, Y  +764.444, Z    +0.000, E1   -69.897, E3 +8011.499}
SPL {X  -129.492, Y  +770.461, Z    +0.000, E1   -69.311, E3 +8018.739}
SPL {X  -125.168, Y  +776.148, Z    +0.000, E1   -68.666, E3 +8025.615}
SPL {X  -122.036, Y  +779.960, Z    +0.000, E1   -68.144, E3 +8030.219}
SPL {X   -80.879, Y  +814.541, Z    +0.000, E1   -55.704, E3 +8151.536}
ENDSPLINE

SPLINE
SPL {X  -125.518, Y  +775.707, Z    +0.000, E1   -52.189, E3 +8323.014}
SPL {X  -144.748, Y  +744.653, Z    +0.000, E1   -45.208, E3 +8341.210}
SPL {X  -153.147, Y  +722.791, Z    +0.000, E1   -36.417, E3 +8347.605}
SPL {X  -157.402, Y  +705.160, Z    +0.000, E1   -26.108, E3 +8350.701}
SPL {X  -159.480, Y  +689.270, Z    +0.000, E1   -14.023, E3 +8352.266}
SPL {X  -159.986, Y  +677.650, Z    +0.000, E1    -3.291, E3 +8352.761}
SPL {X  -159.990, Y  +674.500, Z    +0.000, E1    +0.000, E3 +8352.791}
SPL {X  -159.990, Y  +672.716, Z    +0.000, E1    +3.405, E3 +8352.808}
SPL {X  -159.990, Y  +668.521, Z    +0.000, E1   +13.007, E3 +8352.927}
SPL {X  -159.990, Y  +664.286, Z    +0.000, E1   +23.338, E3 +8353.158}
SPL {X  -159.990, Y  +658.431, Z    +0.000, E1   +35.998, E3 +8353.653}
SPL {X  -159.990, Y  +650.524, Z    +0.000, E1   +48.779, E3 +8354.641}
SPL {X  -159.990, Y  +641.022, Z    +0.000, E1   +57.726, E3 +8356.508}
SPL {X  -159.990, Y  +617.987, Z    +0.000, E1   +67.134, E3 +8362.404}
SPL {X  -159.990, Y  +532.407, Z    +0.000, E1   +73.084, E3 +8393.310}
SPL {X  -159.990, Y  +390.607, Z    +0.000, E1   +73.632, E3 +8464.847}
SPL {X  -159.886, Y  +371.742, Z    +0.000, E1   +73.650, E3 +8476.633}
SPL {X  -157.928, Y  +351.899, Z    +0.000, E1   +73.451, E3 +8491.067}
ENDSPLINE

SPLINE
SPL {X  -159.990, Y  +380.170, Z    +0.000, E1   +69.785, E3 +8507.207}
ENDSPLINE

SPLINE
SPL {X  -158.227, Y  +353.814, Z    +0.000, E1   +70.663, E3 +8519.101}
SPL {X  -155.560, Y  +340.111, Z    +0.000, E1   +70.976, E3 +8526.123}
SPL {X  -151.918, Y  +327.322, Z    +0.000, E1   +71.266, E3 +8532.466}
SPL {X  -144.697, Y  +309.238, Z    +0.000, E1   +71.848, E3 +8539.416}
SPL {X  -140.298, Y  +300.601, Z    +0.000, E1   +71.461, E3 +8547.703}
SPL {X  -137.001, Y  +294.872, Z    +0.000, E1   +71.048, E3 +8554.212}
SPL {X  -133.301, Y  +289.026, Z    +0.000, E1   +70.567, E3 +8560.998}
SPL {X  -129.603, Y  +283.692, Z    +0.000, E1   +70.051, E3 +8567.298}
SPL {X  -125.807, Y  +278.659, Z    +0.000, E1   +69.508, E3 +8573.257}
SPL {X  -122.086, Y  +274.099, Z    +0.000, E1   +68.932, E3 +8578.634}
SPL {X   -84.117, Y  +241.407, Z    +0.000, E1   +58.224, E3 +8669.517}
ENDSPLINE

SPLINE
SPL {X  -116.986, Y  +268.362, Z    +0.000, E1   +53.233, E3 +8863.432}
SPL {X  -146.319, Y  +312.789, Z    +0.000, E1   +44.152, E3 +8893.899}
SPL {X  -157.053, Y  +346.986, Z    +0.000, E1   +27.437, E3 +8901.930}
SPL {X  -159.518, Y  +365.226, Z    +0.000, E1   +13.562, E3 +8903.795}
SPL {X  -159.976, Y  +375.387, Z    +0.000, E1    +4.229, E3 +8904.231}
SPL {X  -159.990, Y  +379.485, Z    +0.000, E1    +0.028, E3 +8904.276}
SPL {X  -159.990, Y  +381.270, Z    +0.000, E1    -3.383, E3 +8904.293}
SPL {X  -159.990, Y  +386.246, Z    +0.000, E1   -14.704, E3 +8904.450}
SPL {X  -159.990, Y  +394.075, Z    +0.000, E1   -32.836, E3 +8905.011}
SPL {X  -159.990, Y  +405.152, Z    +0.000, E1   -50.697, E3 +8906.435}
SPL {X  -159.990, Y  +423.293, Z    +0.000, E1   -63.280, E3 +8910.437}
SPL {X  -159.990, Y  +493.649, Z    +0.000, E1   -71.671, E3 +8936.141}
SPL {X  -159.990, Y  +662.531, Z    +0.000, E1   -73.010, E3 +9022.964}
SPL {X  -159.805, Y  +684.185, Z    +0.000, E1   -72.979, E3 +9037.248}
SPL {X  -158.295, Y  +699.729, Z    +0.000, E1   -72.830, E3 +9048.918}
SPL {X  -155.857, Y  +712.630, Z    +0.000, E1   -72.572, E3 +9059.847}
SPL {X  -153.206, Y  +722.596, Z    +0.000, E1   -72.287, E3 +9069.028}
SPL {X  -150.445, Y  +730.933, Z    +0.000, E1   -71.979, E3 +9077.238}
SPL {X  -147.389, Y  +738.737, Z    +0.000, E1   -71.634, E3 +9085.311}
SPL {X  -144.044, Y  +746.129, Z    +0.000, E1   -71.236, E3 +9093.305}
SPL {X  -140.684, Y  +752.689, Z    +0.000, E1   -70.820, E3 +9100.681}
SPL {X  -137.335, Y  +758.572, Z    +0.000, E1   -70.388, E3 +9107.488}
SPL {X  -133.651, Y  +764.444, Z    +0.000, E1   -69.897, E3 +9114.440}
SPL {X  -129.492, Y  +770.461, Z    +0.000, E1   -69.311, E3 +9121.680}
SPL {X  -125.168, Y  +776.148, Z    +0.000, E1   -68.666, E3 +9128.557}
SPL {X  -122.036, Y  +779.960, Z    +0.000, E1   -68.144, E3 +9133.160}
SPL {X   -80.879, Y  +814.541, Z    +0.000, E1   -55.704, E3 +9254.478}
ENDSPLINE

SPLINE
SPL {X  -125.518, Y  +775.707, Z    +0.000, E1   -52.189, E3 +9425.955}
SPL {X  -144.748, Y  +744.653, Z    +0.000, E1   -45.208, E3 +9444.151}
SPL {X  -153.147, Y  +722.791, Z    +0.000, E1   -36.417, E3 +9450.547}
SPL {X  -157.402, Y  +705.160, Z    +0.000, E1   -26.108, E3 +9453.642}
SPL {X  -159.480, Y  +689.270, Z    +0.000, E1   -14.023, E3 +9455.208}
SPL {X  -159.986, Y  +677.650, Z    +0.000, E1    -3.291, E3 +9455.702}
SPL {X  -159.990, Y  +674.500, Z    +0.000, E1    +0.000, E3 +9455.732}
SPL {X  -159.990, Y  +672.716, Z    +0.000, E1    +3.405, E3 +9455.749}
SPL {X  -159.990, Y  +668.521, Z    +0.000, E1   +13.007, E3 +9455.868}
SPL {X  -159.990, Y  +664.286, Z    +0.000, E1   +23.338, E3 +9456.099}
SPL {X  -159.990, Y  +658.431, Z    +0.000, E1   +35.998, E3 +9456.594}
SPL {X  -159.990, Y  +650.524, Z    +0.000, E1   +48.779, E3 +9457.582}
SPL {X  -159.990, Y  +641.022, Z    +0.000, E1   +57.726, E3 +9459.449}
SPL {X  -159.990, Y  +617.987, Z    +0.000, E1   +67.134, E3 +9465.345}
SPL {X  -159.990, Y  +532.407, Z    +0.000, E1   +73.084, E3 +9496.252}
SPL {X  -159.990, Y  +390.607, Z    +0.000, E1   +73.632, E3 +9567.788}
SPL {X  -159.886, Y  +371.742, Z    +0.000, E1   +73.650, E3 +9579.574}
SPL {X  -157.928, Y  +351.899, Z    +0.000, E1   +73.451, E3 +9594.008}
ENDSPLINE

SPLINE
SPL {X  -159.990, Y  +380.170, Z    +0.000, E1   +69.785, E3 +9610.148}
ENDSPLINE

SPLINE
SPL {X  -158.227, Y  +353.814, Z    +0.000, E1   +70.663, E3 +9622.042}
SPL {X  -155.560, Y  +340.111, Z    +0.000, E1   +70.976, E3 +9629.064}
SPL {X  -151.918, Y  +327.322, Z    +0.000, E1   +71.266, E3 +9635.407}
SPL {X  -144.697, Y  +309.238, Z    +0.000, E1   +71.848, E3 +9642.357}
SPL {X  -140.298, Y  +300.601, Z    +0.000, E1   +71.461, E3 +9650.644}
SPL {X  -135.903, Y  +293.078, Z    +0.000, E1   +70.930, E3 +9659.182}
SPL {X  -130.487, Y  +284.926, Z    +0.000, E1   +70.202, E3 +9668.741}
SPL {X  -125.807, Y  +278.659, Z    +0.000, E1   +69.508, E3 +9676.198}
SPL {X  -122.967, Y  +275.148, Z    +0.000, E1   +69.053, E3 +9680.367}
SPL {X  -121.236, Y  +273.103, Z    +0.000, E1   +68.779, E3 +9682.752}
SPL {X   -84.117, Y  +241.407, Z    +0.000, E1   +58.224, E3 +9772.458}
ENDSPLINE

SPLINE
SPL {X  -116.986, Y  +268.362, Z    +0.000, E1   +53.233, E3 +9966.374}
SPL {X  -146.319, Y  +312.789, Z    +0.000, E1   +44.152, E3 +9996.840}
SPL {X  -157.053, Y  +346.986, Z    +0.000, E1   +27.437, E3 +10004.871}
SPL {X  -159.518, Y  +365.226, Z    +0.000, E1   +13.562, E3 +10006.736}
SPL {X  -159.976, Y  +375.387, Z    +0.000, E1    +4.229, E3 +10007.172}
SPL {X  -159.990, Y  +379.485, Z    +0.000, E1    +0.028, E3 +10007.217}
SPL {X  -159.990, Y  +381.270, Z    +0.000, E1    -3.383, E3 +10007.234}
SPL {X  -159.990, Y  +384.811, Z    +0.000, E1   -11.531, E3 +10007.324}
SPL {X  -159.990, Y  +388.002, Z    +0.000, E1   -19.281, E3 +10007.474}
SPL {X  -159.990, Y  +394.075, Z    +0.000, E1   -32.836, E3 +10007.952}
SPL {X  -159.990, Y  +405.152, Z    +0.000, E1   -50.697, E3 +10009.377}
SPL {X  -159.990, Y  +423.293, Z    +0.000, E1   -63.280, E3 +10013.378}
SPL {X  -159.990, Y  +493.649, Z    +0.000, E1   -71.671, E3 +10039.082}
SPL {X  -159.990, Y  +662.531, Z    +0.000, E1   -73.010, E3 +10125.905}
SPL {X  -159.805, Y  +684.185, Z    +0.000, E1   -72.979, E3 +10140.189}
SPL {X  -158.295, Y  +699.729, Z    +0.000, E1   -72.830, E3 +10151.859}
SPL {X  -155.857, Y  +712.630, Z    +0.000, E1   -72.572, E3 +10162.788}
SPL {X  -153.206, Y  +722.596, Z    +0.000, E1   -72.287, E3 +10171.969}
SPL {X  -150.445, Y  +730.933, Z    +0.000, E1   -71.979, E3 +10180.179}
SPL {X  -147.389, Y  +738.737, Z    +0.000, E1   -71.634, E3 +10188.252}
SPL {X  -144.044, Y  +746.129, Z    +0.000, E1   -71.236, E3 +10196.247}
SPL {X  -140.684, Y  +752.689, Z    +0.000, E1   -70.820, E3 +10203.622}
SPL {X  -136.099, Y  +760.606, Z    +0.000, E1   -70.253, E3 +10212.777}
SPL {X  -131.456, Y  +767.693, Z    +0.000, E1   -69.587, E3 +10221.289}
SPL {X  -127.440, Y  +773.226, Z    +0.000, E1   -69.006, E3 +10227.973}
SPL {X  -123.127, Y  +778.659, Z    +0.000, E1   -68.349, E3 +10234.515}
SPL {X   -80.879, Y  +814.541, Z    +0.000, E1   -55.704, E3 +10357.419}
ENDSPLINE

SPLINE
SPL {X  -125.518, Y  +775.707, Z    +0.000, E1   -52.189, E3 +10528.896}
SPL {X  -144.748, Y  +744.653, Z    +0.000, E1   -45.208, E3 +10547.092}
SPL {X  -153.147, Y  +722.791, Z    +0.000, E1   -36.417, E3 +10553.488}
SPL {X  -158.456, Y  +698.602, Z    +0.000, E1   -21.523, E3 +10557.334}
SPL {X  -159.738, Y  +685.469, Z    +0.000, E1   -10.595, E3 +10558.388}
SPL {X  -159.986, Y  +677.650, Z    +0.000, E1    -3.291, E3 +10558.643}
SPL {X  -159.990, Y  +674.500, Z    +0.000, E1    +0.000, E3 +10558.673}
SPL {X  -159.990, Y  +672.716, Z    +0.000, E1    +3.405, E3 +10558.690}
SPL {X  -159.990, Y  +668.521, Z    +0.000, E1   +13.007, E3 +10558.809}
SPL {X  -159.990, Y  +664.286, Z    +0.000, E1   +23.338, E3 +10559.040}
SPL {X  -159.990, Y  +658.431, Z    +0.000, E1   +35.998, E3 +10559.535}
SPL {X  -159.990, Y  +650.524, Z    +0.000, E1   +48.779, E3 +10560.524}
SPL {X  -159.990, Y  +641.022, Z    +0.000, E1   +57.726, E3 +10562.391}
SPL {X  -159.990, Y  +617.987, Z    +0.000, E1   +67.134, E3 +10568.286}
SPL {X  -159.990, Y  +532.407, Z    +0.000, E1   +73.084, E3 +10599.193}
SPL {X  -159.990, Y  +390.607, Z    +0.000, E1   +73.632, E3 +10670.729}
SPL {X  -159.886, Y  +371.742, Z    +0.000, E1   +73.650, E3 +10682.516}
SPL {X  -157.928, Y  +351.899, Z    +0.000, E1   +73.451, E3 +10696.949}
ENDSPLINE

SPLINE
SPL {X  -159.990, Y  +380.170, Z    +0.000, E1   +69.785, E3 +10713.089}
ENDSPLINE

SPLINE
SPL {X  -158.227, Y  +353.814, Z    +0.000, E1   +70.663, E3 +10724.983}
SPL {X  -154.257, Y  +335.055, Z    +0.000, E1   +71.089, E3 +10734.611}
SPL {X  -148.153, Y  +317.104, Z    +0.000, E1   +71.658, E3 +10741.756}
SPL {X  -143.479, Y  +306.716, Z    +0.000, E1   +71.847, E3 +10746.830}
SPL {X  -140.298, Y  +300.601, Z    +0.000, E1   +71.461, E3 +10753.586}
SPL {X  -137.001, Y  +294.872, Z    +0.000, E1   +71.048, E3 +10760.094}
SPL {X  -133.301, Y  +289.026, Z    +0.000, E1   +70.567, E3 +10766.880}
SPL {X  -128.648, Y  +282.387, Z    +0.000, E1   +69.939, E3 +10774.696}
SPL {X  -125.063, Y  +277.720, Z    +0.000, E1   +69.378, E3 +10780.271}
SPL {X  -122.086, Y  +274.099, Z    +0.000, E1   +68.932, E3 +10784.517}
SPL {X   -84.117, Y  +241.407, Z    +0.000, E1   +58.224, E3 +10875.399}
ENDSPLINE

SPLINE
SPL {X  -106.708, Y  +258.294, Z    +0.000, E1   +53.789, E3 +11054.186}
SPL {X  -137.973, Y  +296.505, Z    +0.000, E1   +48.844, E3 +11092.966}
SPL {X  -154.359, Y  +335.426, Z    +0.000, E1   +34.338, E3 +11105.862}
SPL {X  -159.279, Y  +362.429, Z    +0.000, E1   +16.013, E3 +11109.462}
SPL {X  -159.976, Y  +375.387, Z    +0.000, E1    +4.229, E3 +11110.113}
SPL {X  -159.990, Y  +379.485, Z    +0.000, E1    +0.028, E3 +11110.158}
SPL {X  -159.990, Y  +381.270, Z    +0.000, E1    -3.383, E3 +11110.175}
SPL {X  -159.990, Y  +386.246, Z    +0.000, E1   -14.704, E3 +11110.333}
SPL {X  -159.990, Y  +394.075, Z    +0.000, E1   -32.836, E3 +11110.894}
SPL {X  -159.990, Y  +405.152, Z    +0.000, E1   -50.697, E3 +11112.318}
SPL {X  -159.990, Y  +423.293, Z    +0.000, E1   -63.280, E3 +11116.319}
SPL {X  -159.990, Y  +493.649, Z    +0.000, E1   -71.671, E3 +11142.023}
SPL {X  -159.990, Y  +662.531, Z    +0.000, E1   -73.010, E3 +11228.846}
SPL {X  -159.805, Y  +684.185, Z    +0.000, E1   -72.979, E3 +11243.130}
SPL {X  -158.739, Y  +696.464, Z    +0.000, E1   -72.862, E3 +11252.249}
SPL {X  -156.417, Y  +710.124, Z    +0.000, E1   -72.650, E3 +11263.472}
SPL {X  -153.206, Y  +722.596, Z    +0.000, E1   -72.287, E3 +11274.910}
SPL {X  -150.445, Y  +730.933, Z    +0.000, E1   -71.979, E3 +11283.121}
SPL {X  -147.389, Y  +738.737, Z    +0.000, E1   -71.634, E3 +11291.193}
SPL {X  -144.044, Y  +746.129, Z    +0.000, E1   -71.236, E3 +11299.188}
SPL {X  -140.684, Y  +752.689, Z    +0.000, E1   -70.820, E3 +11306.563}
SPL {X  -137.335, Y  +758.572, Z    +0.000, E1   -70.388, E3 +11313.370}
SPL {X  -133.651, Y  +764.444, Z    +0.000, E1   -69.897, E3 +11320.322}
SPL {X  -130.650, Y  +768.844, Z    +0.000, E1   -69.455, E3 +11325.644}
SPL {X  -127.440, Y  +773.226, Z    +0.000, E1   -69.006, E3 +11330.914}
SPL {X  -123.127, Y  +778.659, Z    +0.000, E1   -68.349, E3 +11337.456}
SPL {X   -80.879, Y  +814.541, Z    +0.000, E1   -55.704, E3 +11460.360}
ENDSPLINE

SPLINE
SPL {X  -125.518, Y  +775.707, Z    +0.000, E1   -52.189, E3 +11631.837}
SPL {X  -150.797, Y  +729.951, Z    +0.000, E1   -39.777, E3 +11654.572}
SPL {X  -158.456, Y  +698.602, Z    +0.000, E1   -21.523, E3 +11660.275}
SPL {X  -159.738, Y  +685.469, Z    +0.000, E1   -10.595, E3 +11661.329}
SPL {X  -159.986, Y  +677.650, Z    +0.000, E1    -3.291, E3 +11661.584}
SPL {X  -159.990, Y  +674.500, Z    +0.000, E1    +0.000, E3 +11661.615}
SPL {X  -159.990, Y  +672.716, Z    +0.000, E1    +3.405, E3 +11661.631}
SPL {X  -159.990, Y  +668.521, Z    +0.000, E1   +13.007, E3 +11661.750}
SPL {X  -159.990, Y  +662.839, Z    +0.000, E1   +26.519, E3 +11662.093}
SPL {X  -159.990, Y  +653.836, Z    +0.000, E1   +43.967, E3 +11663.023}
SPL {X  -159.990, Y  +641.022, Z    +0.000, E1   +57.726, E3 +11665.332}
SPL {X  -159.990, Y  +617.987, Z    +0.000, E1   +67.134, E3 +11671.227}
SPL {X  -159.990, Y  +532.407, Z    +0.000, E1   +73.084, E3 +11702.134}
SPL {X  -159.990, Y  +382.957, Z    +0.000, E1   +73.647, E3 +11778.394}
SPL {X  -159.615, Y  +366.548, Z    +0.000, E1   +73.602, E3 +11789.036}
SPL {X  -157.928, Y  +351.899, Z    +0.000, E1   +73.451, E3 +11799.890}
ENDSPLINE

SPLINE
SPL {X  -159.990, Y  +380.170, Z    +0.000, E1   +69.785, E3 +11816.031}
ENDSPLINE

SPLINE
SPL {X  -158.227, Y  +353.814, Z    +0.000, E1   +70.663, E3 +11827.924}
SPL {X  -154.257, Y  +335.055, Z    +0.000, E1   +71.089, E3 +11837.552}
SPL {X  -148.153, Y  +317.104, Z    +0.000, E1   +71.658, E3 +11844.698}
SPL {X  -143.479, Y  +306.716, Z    +0.000, E1   +71.847, E3 +11849.771}
SPL {X  -140.298, Y  +300.601, Z    +0.000, E1   +71.461, E3 +11856.527}
SPL {X  -137.001, Y  +294.872, Z    +0.000, E1   +71.048, E3 +11863.035}
SPL {X  -133.301, Y  +289.026, Z    +0.000, E1   +70.567, E3 +11869.822}
SPL {X  -129.603, Y  +283.692, Z    +0.000, E1   +70.051, E3 +11876.122}
SPL {X  -125.807, Y  +278.659, Z    +0.000, E1   +69.508, E3 +11882.080}
SPL {X  -122.086, Y  +274.099, Z    +0.000, E1   +68.932, E3 +11887.458}
SPL {X   -84.117, Y  +241.407, Z    +0.000, E1   +58.224, E3 +11978.341}
ENDSPLINE

SPLINE
SPL {X  -116.986, Y  +268.362, Z    +0.000, E1   +53.233, E3 +12172.256}
SPL {X  -146.319, Y  +312.789, Z    +0.000, E1   +44.152, E3 +12202.722}
SPL {X  -157.053, Y  +346.986, Z    +0.000, E1   +27.437, E3 +12210.753}
SPL {X  -159.518, Y  +365.226, Z    +0.000, E1   +13.562, E3 +12212.619}
SPL {X  -159.976, Y  +375.387, Z    +0.000, E1    +4.229, E3 +12213.054}
SPL {X  -159.990, Y  +379.485, Z    +0.000, E1    +0.028, E3 +12213.099}
SPL {X  -159.990, Y  +381.270, Z    +0.000, E1    -3.383, E3 +12213.117}
SPL {X  -159.990, Y  +384.811, Z    +0.000, E1   -11.531, E3 +12213.207}
SPL {X  -159.990, Y  +390.180, Z    +0.000, E1   -24.142, E3 +12213.510}
SPL {X  -159.990, Y  +397.074, Z    +0.000, E1   -39.012, E3 +12214.120}
SPL {X  -159.990, Y  +405.152, Z    +0.000, E1   -50.697, E3 +12215.259}
SPL {X  -159.990, Y  +423.293, Z    +0.000, E1   -63.280, E3 +12219.260}
SPL {X  -159.990, Y  +493.649, Z    +0.000, E1   -71.671, E3 +12244.964}
SPL {X  -159.990, Y  +662.531, Z    +0.000, E1   -73.010, E3 +12331.787}
SPL {X  -159.805, Y  +684.185, Z    +0.000, E1   -72.979, E3 +12346.071}
SPL {X  -158.739, Y  +696.464, Z    +0.000, E1   -72.862, E3 +12355.190}
SPL {X  -156.417, Y  +710.124, Z    +0.000, E1   -72.650, E3 +12366.413}
SPL {X  -153.206, Y  +722.596, Z    +0.000, E1   -72.287, E3 +12377.851}
SPL {X  -150.445, Y  +730.933, Z    +0.000, E1   -71.979, E3 +12386.062}
SPL {X  -147.389, Y  +738.737, Z    +0.000, E1   -71.634, E3 +12394.135}
SPL {X  -144.044, Y  +746.129, Z    +0.000, E1   -71.236, E3 +12402.129}
SPL {X  -140.684, Y  +752.689, Z    +0.000, E1   -70.820, E3 +12409.504}
SPL {X  -137.335, Y  +758.572, Z    +0.000, E1   -70.388, E3 +12416.311}
SPL {X  -134.566, Y  +763.037, Z    +0.000, E1   -70.007, E3 +12421.608}
SPL {X  -131.456, Y  +767.693, Z    +0.000, E1   -69.587, E3 +12427.171}
SPL {X  -127.440, Y  +773.226, Z    +0.000, E1   -69.006, E3 +12433.855}
SPL {X  -123.127, Y  +778.659, Z    +0.000, E1   -68.349, E3 +12440.397}
SPL {X   -80.879, Y  +814.541, Z    +0.000, E1   -55.704, E3 +12563.301}
ENDSPLINE

SPLINE
SPL {X  -125.518, Y  +775.707, Z    +0.000, E1   -52.189, E3 +12734.779}
SPL {X  -144.748, Y  +744.653, Z    +0.000, E1   -45.208, E3 +12752.974}
SPL {X  -153.147, Y  +722.791, Z    +0.000, E1   -36.417, E3 +12759.370}
SPL {X  -157.402, Y  +705.160, Z    +0.000, E1   -26.108, E3 +12762.465}
SPL {X  -159.480, Y  +689.270, Z    +0.000, E1   -14.023, E3 +12764.031}
SPL {X  -159.986, Y  +677.650, Z    +0.000, E1    -3.291, E3 +12764.525}
SPL {X  -159.990, Y  +674.500, Z    +0.000, E1    +0.000, E3 +12764.556}
SPL {X  -159.990, Y  +672.716, Z    +0.000, E1    +3.405, E3 +12764.572}
SPL {X  -159.990, Y  +668.521, Z    +0.000, E1   +13.007, E3 +12764.691}
SPL {X  -159.990, Y  +662.839, Z    +0.000, E1   +26.519, E3 +12765.034}
SPL {X  -159.990, Y  +653.836, Z    +0.000, E1   +43.967, E3 +12765.964}
SPL {X  -159.990, Y  +641.022, Z    +0.000, E1   +57.726, E3 +12768.273}
SPL {X  -159.990, Y  +617.987, Z    +0.000, E1   +67.134, E3 +12774.168}
SPL {X  -159.990, Y  +532.407, Z    +0.000, E1   +73.084, E3 +12805.075}
SPL {X  -159.990, Y  +382.957, Z    +0.000, E1   +73.647, E3 +12881.335}
SPL {X  -159.615, Y  +366.548, Z    +0.000, E1   +73.602, E3 +12891.977}
SPL {X  -157.928, Y  +351.899, Z    +0.000, E1   +73.451, E3 +12902.832}
ENDSPLINE

SPLINE
SPL {X  -159.990, Y  +380.170, Z    +0.000, E1   +69.785, E3 +12918.972}
ENDSPLINE

SPLINE
SPL {X  -158.227, Y  +353.814, Z    +0.000, E1   +70.663, E3 +12930.865}
SPL {X  -155.560, Y  +340.111, Z    +0.000, E1   +70.976, E3 +12937.887}
SPL {X  -151.918, Y  +327.322, Z    +0.000, E1   +71.266, E3 +12944.231}
SPL {X  -144.697, Y  +309.238, Z    +0.000, E1   +71.848, E3 +12951.181}
SPL {X  -140.298, Y  +300.601, Z    +0.000, E1   +71.461, E3 +12959.468}
SPL {X  -137.001, Y  +294.872, Z    +0.000, E1   +71.048, E3 +12965.976}
SPL {X  -133.301, Y  +289.026, Z    +0.000, E1   +70.567, E3 +12972.763}
SPL {X  -129.603, Y  +283.692, Z    +0.000, E1   +70.051, E3 +12979.063}
SPL {X  -125.807, Y  +278.659, Z    +0.000, E1   +69.508, E3 +12985.022}
SPL {X  -122.086, Y  +274.099, Z    +0.000, E1   +68.932, E3 +12990.399}
SPL {X   -84.117, Y  +241.407, Z    +0.000, E1   +58.224, E3 +13081.282}
ENDSPLINE

SPLINE
SPL {X  -106.708, Y  +258.294, Z    +0.000, E1   +53.789, E3 +13260.069}
SPL {X  -137.973, Y  +296.505, Z    +0.000, E1   +48.844, E3 +13298.849}
SPL {X  -154.359, Y  +335.426, Z    +0.000, E1   +34.338, E3 +13311.745}
SPL {X  -159.279, Y  +362.429, Z    +0.000, E1   +16.013, E3 +13315.345}
SPL {X  -159.976, Y  +375.387, Z    +0.000, E1    +4.229, E3 +13315.996}
SPL {X  -159.990, Y  +379.485, Z    +0.000, E1    +0.028, E3 +13316.041}
SPL {X  -159.990, Y  +381.270, Z    +0.000, E1    -3.383, E3 +13316.058}
SPL {X  -159.990, Y  +386.246, Z    +0.000, E1   -14.704, E3 +13316.215}
SPL {X  -159.990, Y  +394.075, Z    +0.000, E1   -32.836, E3 +13316.776}
SPL {X  -159.990, Y  +405.152, Z    +0.000, E1   -50.697, E3 +13318.200}
SPL {X  -159.990, Y  +423.293, Z    +0.000, E1   -63.280, E3 +13322.201}
SPL {X  -159.990, Y  +493.649, Z    +0.000, E1   -71.671, E3 +13347.905}
SPL {X  -159.990, Y  +662.531, Z    +0.000, E1   -73.010, E3 +13434.728}
SPL {X  -159.805, Y  +684.185, Z    +0.000, E1   -72.979, E3 +13449.012}
SPL {X  -158.739, Y  +696.464, Z    +0.000, E1   -72.862, E3 +13458.131}
SPL {X  -156.417, Y  +710.124, Z    +0.000, E1   -72.650, E3 +13469.355}
SPL {X  -153.206, Y  +722.596, Z    +0.000, E1   -72.287, E3 +13480.793}
SPL {X  -150.445, Y  +730.933, Z    +0.000, E1   -71.979, E3 +13489.003}
SPL {X  -147.389, Y  +738.737, Z    +0.000, E1   -71.634, E3 +13497.076}
SPL {X  -144.044, Y  +746.129, Z    +0.000, E1   -71.236, E3 +13505.070}
SPL {X  -140.684, Y  +752.689, Z    +0.000, E1   -70.820, E3 +13512.445}
SPL {X  -137.335, Y  +758.572, Z    +0.000, E1   -70.388, E3 +13519.253}
SPL {X  -133.651, Y  +764.444, Z    +0.000, E1   -69.897, E3 +13526.205}
SPL {X  -129.492, Y  +770.461, Z    +0.000, E1   -69.311, E3 +13533.445}
SPL {X  -125.168, Y  +776.148, Z    +0.000, E1   -68.666, E3 +13540.321}
SPL {X  -122.036, Y  +779.960, Z    +0.000, E1   -68.144, E3 +13544.925}
SPL {X   -80.879, Y  +814.541, Z    +0.000, E1   -55.704, E3 +13666.242}
ENDSPLINE

SPLINE
SPL {X  -125.518, Y  +775.707, Z    +0.000, E1   -52.189, E3 +13837.720}
SPL {X  -144.748, Y  +744.653, Z    +0.000, E1   -45.208, E3 +13855.916}
SPL {X  -153.147, Y  +722.791, Z    +0.000, E1   -36.417, E3 +13862.311}
SPL {X  -157.402, Y  +705.160, Z    +0.000, E1   -26.108, E3 +13865.407}
SPL {X  -159.480, Y  +689.270, Z    +0.000, E1   -14.023, E3 +13866.972}
SPL {X  -159.986, Y  +677.650, Z    +0.000, E1    -3.291, E3 +13867.467}
SPL {X  -159.990, Y  +674.500, Z    +0.000, E1    +0.000, E3 +13867.497}
SPL {X  -159.990, Y  +672.716, Z    +0.000, E1    +3.405, E3 +13867.513}
SPL {X  -159.990, Y  +668.521, Z    +0.000, E1   +13.007, E3 +13867.633}
SPL {X  -159.990, Y  +664.286, Z    +0.000, E1   +23.338, E3 +13867.864}
SPL {X  -159.990, Y  +658.431, Z    +0.000, E1   +35.998, E3 +13868.359}
SPL {X  -159.990, Y  +650.524, Z    +0.000, E1   +48.779, E3 +13869.347}
SPL {X  -159.990, Y  +641.022, Z    +0.000, E1   +57.726, E3 +13871.214}
SPL {X  -159.990, Y  +617.987, Z    +0.000, E1   +67.134, E3 +13877.110}
SPL {X  -159.990, Y  +532.407, Z    +0.000, E1   +73.084, E3 +13908.016}
SPL {X  -159.990, Y  +390.607, Z    +0.000, E1   +73.632, E3 +13979.552}
SPL {X  -159.886, Y  +371.742, Z    +0.000, E1   +73.650, E3 +13991.339}
SPL {X  -157.928, Y  +351.899, Z    +0.000, E1   +73.451, E3 +14005.773}
ENDSPLINE

SPLINE
SPL {X  -159.990, Y  +380.170, Z    +0.000, E1   +69.785, E3 +14021.913}
ENDSPLINE

SPLINE
SPL {X  -158.227, Y  +353.814, Z    +0.000, E1   +70.663, E3 +14033.806}
SPL {X  -155.560, Y  +340.111, Z    +0.000, E1   +70.976, E3 +14040.829}
SPL {X  -151.918, Y  +327.322, Z    +0.000, E1   +71.266, E3 +14047.172}
SPL {X  -144.697, Y  +309.238, Z    +0.000, E1   +71.848, E3 +14054.122}
SPL {X  -140.298, Y  +300.601, Z    +0.000, E1   +71.461, E3 +14062.409}
SPL {X  -137.001, Y  +294.872, Z    +0.000, E1   +71.048, E3 +14068.917}
SPL {X  -133.301, Y  +289.026, Z    +0.000, E1   +70.567, E3 +14075.704}
SPL {X  -129.603, Y  +283.692, Z    +0.000, E1   +70.051, E3 +14082.004}
SPL {X  -125.807, Y  +278.659, Z    +0.000, E1   +69.508, E3 +14087.963}
SPL {X  -122.086, Y  +274.099, Z    +0.000, E1   +68.932, E3 +14093.340}
SPL {X   -84.117, Y  +241.407, Z    +0.000, E1   +58.224, E3 +14184.223}
ENDSPLINE

SPLINE
SPL {X  -116.986, Y  +268.362, Z    +0.000, E1   +53.233, E3 +14378.138}
SPL {X  -146.319, Y  +312.789, Z    +0.000, E1   +44.152, E3 +14408.604}
SPL {X  -157.053, Y  +346.986, Z    +0.000, E1   +27.437, E3 +14416.636}
SPL {X  -159.518, Y  +365.226, Z    +0.000, E1   +13.562, E3 +14418.501}
SPL {X  -159.976, Y  +375.387, Z    +0.000, E1    +4.229, E3 +14418.937}
SPL {X  -159.990, Y  +379.485, Z    +0.000, E1    +0.028, E3 +14418.982}
SPL {X  -159.990, Y  +381.270, Z    +0.000, E1    -3.383, E3 +14418.999}
SPL {X  -159.990, Y  +386.246, Z    +0.000, E1   -14.704, E3 +14419.156}
SPL {X  -159.990, Y  +394.075, Z    +0.000, E1   -32.836, E3 +14419.717}
SPL {X  -159.990, Y  +405.152, Z    +0.000, E1   -50.697, E3 +14421.141}
SPL {X  -159.990, Y  +423.293, Z    +0.000, E1   -63.280, E3 +14425.143}
SPL {X  -159.990, Y  +493.649, Z    +0.000, E1   -71.671, E3 +14450.847}
SPL {X  -159.990, Y  +662.531, Z    +0.000, E1   -73.010, E3 +14537.670}
SPL {X  -159.805, Y  +684.185, Z    +0.000, E1   -72.979, E3 +14551.954}
SPL {X  -158.295, Y  +699.729, Z    +0.000, E1   -72.830, E3 +14563.624}
SPL {X  -155.857, Y  +712.630, Z    +0.000, E1   -72.572, E3 +14574.553}
SPL {X  -153.206, Y  +722.596, Z    +0.000, E1   -72.287, E3 +14583.734}
SPL {X  -150.445, Y  +730.933, Z    +0.000, E1   -71.979, E3 +14591.944}
SPL {X  -147.389, Y  +738.737, Z    +0.000, E1   -71.634, E3 +14600.017}
SPL {X  -144.044, Y  +746.129, Z    +0.000, E1   -71.236, E3 +14608.011}
SPL {X  -140.684, Y  +752.689, Z    +0.000, E1   -70.820, E3 +14615.387}
SPL {X  -136.099, Y  +760.606, Z    +0.000, E1   -70.253, E3 +14624.542}
SPL {X  -131.456, Y  +767.693, Z    +0.000, E1   -69.587, E3 +14633.054}
SPL {X  -128.507, Y  +771.803, Z    +0.000, E1   -69.145, E3 +14638.036}
SPL {X  -125.168, Y  +776.148, Z    +0.000, E1   -68.666, E3 +14643.262}
SPL {X  -122.036, Y  +779.960, Z    +0.000, E1   -68.144, E3 +14647.866}
SPL {X   -80.879, Y  +814.541, Z    +0.000, E1   -55.704, E3 +14769.184}
ENDSPLINE

SPLINE
SPL {X  -125.518, Y  +775.707, Z    +0.000, E1   -52.189, E3 +14940.661}
SPL {X  -150.797, Y  +729.951, Z    +0.000, E1   -39.777, E3 +14963.396}
SPL {X  -158.456, Y  +698.602, Z    +0.000, E1   -21.523, E3 +14969.099}
SPL {X  -159.738, Y  +685.469, Z    +0.000, E1   -10.595, E3 +14970.153}
SPL {X  -159.986, Y  +677.650, Z    +0.000, E1    -3.291, E3 +14970.408}
SPL {X  -159.990, Y  +674.500, Z    +0.000, E1    +0.000, E3 +14970.438}
SPL {X  -159.990, Y  +672.716, Z    +0.000, E1    +3.405, E3 +14970.455}
SPL {X  -159.990, Y  +668.521, Z    +0.000, E1   +13.007, E3 +14970.574}
SPL {X  -159.990, Y  +662.839, Z    +0.000, E1   +26.519, E3 +14970.916}
SPL {X  -159.990, Y  +653.836, Z    +0.000, E1   +43.967, E3 +14971.846}
SPL {X  -159.990, Y  +641.022, Z    +0.000, E1   +57.726, E3 +14974.155}
SPL {X  -159.990, Y  +617.987, Z    +0.000, E1   +67.134, E3 +14980.051}
SPL {X  -159.990, Y  +532.407, Z    +0.000, E1   +73.084, E3 +15010.957}
SPL {X  -159.990, Y  +382.957, Z    +0.000, E1   +73.647, E3 +15087.217}
SPL {X  -159.615, Y  +366.548, Z    +0.000, E1   +73.602, E3 +15097.859}
SPL {X  -157.928, Y  +351.899, Z    +0.000, E1   +73.451, E3 +15108.714}
ENDSPLINE

SPLINE
SPL {X  -159.990, Y  +380.170, Z    +0.000, E1   +69.785, E3 +15124.854}
ENDSPLINE

SPLINE
SPL {X  -158.227, Y  +353.814, Z    +0.000, E1   +70.663, E3 +15136.748}
SPL {X  -154.257, Y  +335.055, Z    +0.000, E1   +71.089, E3 +15146.376}
SPL {X  -148.153, Y  +317.104, Z    +0.000, E1   +71.658, E3 +15153.521}
SPL {X  -143.479, Y  +306.716, Z    +0.000, E1   +71.847, E3 +15158.595}
SPL {X  -140.298, Y  +300.601, Z    +0.000, E1   +71.461, E3 +15165.350}
SPL {X  -137.001, Y  +294.872, Z    +0.000, E1   +71.048, E3 +15171.859}
SPL {X  -133.301, Y  +289.026, Z    +0.000, E1   +70.567, E3 +15178.645}
SPL {X  -128.648, Y  +282.387, Z    +0.000, E1   +69.939, E3 +15186.460}
SPL {X  -125.063, Y  +277.720, Z    +0.000, E1   +69.378, E3 +15192.036}
SPL {X  -122.086, Y  +274.099, Z    +0.000, E1   +68.932, E3 +15196.281}
SPL {X   -84.117, Y  +241.407, Z    +0.000, E1   +58.224, E3 +15287.164}
ENDSPLINE

SPLINE
SPL {X  -106.708, Y  +258.294, Z    +0.000, E1   +53.789, E3 +15465.951}
SPL {X  -137.973, Y  +296.505, Z    +0.000, E1   +48.844, E3 +15504.731}
SPL {X  -150.692, Y  +323.752, Z    +0.000, E1   +39.895, E3 +15515.097}
SPL {X  -157.053, Y  +346.986, Z    +0.000, E1   +27.437, E3 +15519.577}
SPL {X  -159.518, Y  +365.226, Z    +0.000, E1   +13.562, E3 +15521.442}
SPL {X  -159.976, Y  +375.387, Z    +0.000, E1    +4.229, E3 +15521.878}
SPL {X  -159.990, Y  +379.485, Z    +0.000, E1    +0.028, E3 +15521.923}
SPL {X  -159.990, Y  +381.270, Z    +0.000, E1    -3.383, E3 +15521.940}
SPL {X  -159.990, Y  +386.246, Z    +0.000, E1   -14.704, E3 +15522.098}
SPL {X  -159.990, Y  +394.075, Z    +0.000, E1   -32.836, E3 +15522.658}
SPL {X  -159.990, Y  +405.152, Z    +0.000, E1   -50.697, E3 +15524.082}
SPL {X  -159.990, Y  +423.293, Z    +0.000, E1   -63.280, E3 +15528.084}
SPL {X  -159.990, Y  +493.649, Z    +0.000, E1   -71.671, E3 +15553.788}
SPL {X  -159.990, Y  +662.531, Z    +0.000, E1   -73.010, E3 +15640.611}
SPL {X  -159.805, Y  +684.185, Z    +0.000, E1   -72.979, E3 +15654.895}
SPL {X  -158.295, Y  +699.729, Z    +0.000, E1   -72.830, E3 +15666.565}
SPL {X  -155.857, Y  +712.630, Z    +0.000, E1   -72.572, E3 +15677.494}
SPL {X  -153.206, Y  +722.596, Z    +0.000, E1   -72.287, E3 +15686.675}
SPL {X  -150.445, Y  +730.933, Z    +0.000, E1   -71.979, E3 +15694.885}
SPL {X  -147.389, Y  +738.737, Z    +0.000, E1   -71.634, E3 +15702.958}
SPL {X  -144.044, Y  +746.129, Z    +0.000, E1   -71.236, E3 +15710.952}
SPL {X  -140.684, Y  +752.689, Z    +0.000, E1   -70.820, E3 +15718.328}
SPL {X  -136.099, Y  +760.606, Z    +0.000, E1   -70.253, E3 +15727.483}
SPL {X  -131.456, Y  +767.693, Z    +0.000, E1   -69.587, E3 +15735.995}
SPL {X  -128.507, Y  +771.803, Z    +0.000, E1   -69.145, E3 +15740.977}
SPL {X  -125.168, Y  +776.148, Z    +0.000, E1   -68.666, E3 +15746.204}
SPL {X  -122.036, Y  +779.960, Z    +0.000, E1   -68.144, E3 +15750.807}
SPL {X   -80.879, Y  +814.541, Z    +0.000, E1   -55.704, E3 +15872.125}
ENDSPLINE

SPLINE
SPL {X  -125.518, Y  +775.707, Z    +0.000, E1   -52.189, E3 +16043.602}
SPL {X  -150.797, Y  +729.951, Z    +0.000, E1   -39.777, E3 +16066.337}
SPL {X  -158.456, Y  +698.602, Z    +0.000, E1   -21.523, E3 +16072.040}
SPL {X  -159.738, Y  +685.469, Z    +0.000, E1   -10.595, E3 +16073.094}
SPL {X  -159.986, Y  +677.650, Z    +0.000, E1    -3.291, E3 +16073.349}
SPL {X  -159.990, Y  +674.500, Z    +0.000, E1    +0.000, E3 +16073.379}
SPL {X  -159.990, Y  +672.716, Z    +0.000, E1    +3.405, E3 +16073.396}
SPL {X  -159.990, Y  +668.521, Z    +0.000, E1   +13.007, E3 +16073.515}
SPL {X  -159.990, Y  +662.839, Z    +0.000, E1   +26.519, E3 +16073.857}
SPL {X  -159.990, Y  +653.836, Z    +0.000, E1   +43.967, E3 +16074.787}
SPL {X  -159.990, Y  +641.022, Z    +0.000, E1   +57.726, E3 +16077.096}
SPL {X  -159.990, Y  +617.987, Z    +0.000, E1   +67.134, E3 +16082.992}
SPL {X  -159.990, Y  +532.407, Z    +0.000, E1   +73.084, E3 +16113.899}
SPL {X  -159.990, Y  +390.607, Z    +0.000, E1   +73.632, E3 +16185.435}
SPL {X  -159.886, Y  +371.742, Z    +0.000, E1   +73.650, E3 +16197.222}
SPL {X  -157.928, Y  +351.899, Z    +0.000, E1   +73.451, E3 +16211.655}
ENDSPLINE

SPLINE
SPL {X  -159.990, Y  +387.996, Z    +0.000, E1   +69.509, E3 +16224.085}
ENDSPLINE

SPLINE
SPL {X  -159.889, Y  +371.819, Z    +0.000, E1   +70.046, E3 +16231.812}
SPL {X  -158.227, Y  +353.814, Z    +0.000, E1   +70.663, E3 +16239.689}
SPL {X  -154.257, Y  +335.055, Z    +0.000, E1   +71.089, E3 +16249.317}
SPL {X  -148.153, Y  +317.104, Z    +0.000, E1   +71.658, E3 +16256.462}
SPL {X  -143.479, Y  +306.716, Z    +0.000, E1   +71.847, E3 +16261.536}
SPL {X  -140.298, Y  +300.601, Z    +0.000, E1   +71.461, E3 +16268.292}
SPL {X  -135.903, Y  +293.078, Z    +0.000, E1   +70.930, E3 +16276.829}
SPL {X  -130.487, Y  +284.926, Z    +0.000, E1   +70.202, E3 +16286.388}
SPL {X  -125.807, Y  +278.659, Z    +0.000, E1   +69.508, E3 +16293.845}
SPL {X  -122.086, Y  +274.099, Z    +0.000, E1   +68.932, E3 +16299.223}
SPL {X   -84.117, Y  +241.407, Z    +0.000, E1   +58.224, E3 +16390.105}
ENDSPLINE

SPLINE
SPL {X  -106.708, Y  +258.294, Z    +0.000, E1   +53.789, E3 +16568.892}
SPL {X  -137.973, Y  +296.505, Z    +0.000, E1   +48.844, E3 +16607.672}
SPL {X  -154.359, Y  +335.426, Z    +0.000, E1   +34.338, E3 +16620.568}
SPL {X  -159.279, Y  +362.429, Z    +0.000, E1   +16.013, E3 +16624.168}
SPL {X  -159.976, Y  +375.387, Z    +0.000, E1    +4.229, E3 +16624.819}
SPL {X  -159.990, Y  +379.485, Z    +0.000, E1    +0.028, E3 +16624.864}
SPL {X  -159.990, Y  +381.270, Z    +0.000, E1    -3.383, E3 +16624.881}
SPL {X  -159.990, Y  +384.811, Z    +0.000, E1   -11.531, E3 +16624.971}
SPL {X  -159.990, Y  +390.180, Z    +0.000, E1   -24.142, E3 +16625.274}
SPL {X  -159.990, Y  +397.074, Z    +0.000, E1   -39.012, E3 +16625.884}
SPL {X  -159.990, Y  +405.152, Z    +0.000, E1   -50.697, E3 +16627.024}
SPL {X  -159.990, Y  +423.293, Z    +0.000, E1   -63.280, E3 +16631.025}
SPL {X  -159.990, Y  +493.649, Z    +0.000, E1   -71.671, E3 +16656.729}
SPL {X  -159.990, Y  +662.531, Z    +0.000, E1   -73.010, E3 +16743.552}
SPL {X  -159.805, Y  +684.185, Z    +0.000, E1   -72.979, E3 +16757.836}
SPL {X  -158.295, Y  +699.729, Z    +0.000, E1   -72.830, E3 +16769.506}
SPL {X  -155.857, Y  +712.630, Z    +0.000, E1   -72.572, E3 +16780.435}
SPL {X  -153.206, Y  +722.596, Z    +0.000, E1   -72.287, E3 +16789.616}
SPL {X  -150.445, Y  +730.933, Z    +0.000, E1   -71.979, E3 +16797.827}
SPL {X  -147.389, Y  +738.737, Z    +0.000, E1   -71.634, E3 +16805.899}
SPL {X  -144.044, Y  +746.129, Z    +0.000, E1   -71.236, E3 +16813.894}
SPL {X  -140.684, Y  +752.689, Z    +0.000, E1   -70.820, E3 +16821.269}
SPL {X  -136.099, Y  +760.606, Z    +0.000, E1   -70.253, E3 +16830.424}
SPL {X  -131.456, Y  +767.693, Z    +0.000, E1   -69.587, E3 +16838.936}
SPL {X  -128.507, Y  +771.803, Z    +0.000, E1   -69.145, E3 +16843.918}
SPL {X  -125.168, Y  +776.148, Z    +0.000, E1   -68.666, E3 +16849.145}
SPL {X  -122.036, Y  +779.960, Z    +0.000, E1   -68.144, E3 +16853.748}
SPL {X   -80.879, Y  +814.541, Z    +0.000, E1   -55.704, E3 +16975.066}
ENDSPLINE

SPLINE
SPL {X  -125.518, Y  +775.707, Z    +0.000, E1   -52.189, E3 +17146.543}
SPL {X  -144.748, Y  +744.653, Z    +0.000, E1   -45.208, E3 +17164.739}
SPL {X  -153.147, Y  +722.791, Z    +0.000, E1   -36.417, E3 +17171.135}
SPL {X  -158.456, Y  +698.602, Z    +0.000, E1   -21.523, E3 +17174.981}
SPL {X  -159.738, Y  +685.469, Z    +0.000, E1   -10.595, E3 +17176.035}
SPL {X  -159.986, Y  +677.650, Z    +0.000, E1    -3.291, E3 +17176.290}
SPL {X  -159.990, Y  +674.500, Z    +0.000, E1    +0.000, E3 +17176.320}
SPL {X  -159.990, Y  +672.716, Z    +0.000, E1    +3.405, E3 +17176.337}
SPL {X  -159.990, Y  +668.521, Z    +0.000, E1   +13.007, E3 +17176.456}
SPL {X  -159.990, Y  +664.286, Z    +0.000, E1   +23.338, E3 +17176.688}
SPL {X  -159.990, Y  +658.431, Z    +0.000, E1   +35.998, E3 +17177.182}
SPL {X  -159.990, Y  +650.524, Z    +0.000, E1   +48.779, E3 +17178.171}
SPL {X  -159.990, Y  +641.022, Z    +0.000, E1   +57.726, E3 +17180.038}
SPL {X  -159.990, Y  +617.987, Z    +0.000, E1   +67.134, E3 +17185.933}
SPL {X  -159.990, Y  +532.407, Z    +0.000, E1   +73.084, E3 +17216.840}
SPL {X  -159.990, Y  +382.957, Z    +0.000, E1   +73.647, E3 +17293.099}
SPL {X  -159.615, Y  +366.548, Z    +0.000, E1   +73.602, E3 +17303.742}
SPL {X  -157.928, Y  +351.899, Z    +0.000, E1   +73.451, E3 +17314.596}
ENDSPLINE

SPLINE
SPL {X  -159.990, Y  +380.170, Z    +0.000, E1   +69.785, E3 +17330.736}
ENDSPLINE

SPLINE
SPL {X  -158.227, Y  +353.814, Z    +0.000, E1   +70.663, E3 +17342.630}
SPL {X  -155.560, Y  +340.111, Z    +0.000, E1   +70.976, E3 +17349.652}
SPL {X  -151.918, Y  +327.322, Z    +0.000, E1   +71.266, E3 +17355.996}
SPL {X  -144.697, Y  +309.238, Z    +0.000, E1   +71.848, E3 +17362.945}
SPL {X  -140.298, Y  +300.601, Z    +0.000, E1   +71.461, E3 +17371.233}
SPL {X  -137.001, Y  +294.872, Z    +0.000, E1   +71.048, E3 +17377.741}
SPL {X  -133.301, Y  +289.026, Z    +0.000, E1   +70.567, E3 +17384.527}
SPL {X  -128.648, Y  +282.387, Z    +0.000, E1   +69.939, E3 +17392.343}
SPL {X  -125.063, Y  +277.720, Z    +0.000, E1   +69.378, E3 +17397.918}
SPL {X  -122.086, Y  +274.099, Z    +0.000, E1   +68.932, E3 +17402.164}
SPL {X   -84.117, Y  +241.407, Z    +0.000, E1   +58.224, E3 +17493.046}
ENDSPLINE

SPLINE
SPL {X  -106.708, Y  +258.294, Z    +0.000, E1   +53.789, E3 +17671.833}
SPL {X  -137.973, Y  +296.505, Z    +0.000, E1   +48.844, E3 +17710.613}
SPL {X  -154.359, Y  +335.426, Z    +0.000, E1   +34.338, E3 +17723.509}
SPL {X  -159.279, Y  +362.429, Z    +0.000, E1   +16.013, E3 +17727.110}
SPL {X  -159.976, Y  +375.387, Z    +0.000, E1    +4.229, E3 +17727.760}
SPL {X  -159.990, Y  +379.485, Z    +0.000, E1    +0.028, E3 +17727.805}
SPL {X  -159.990, Y  +381.270, Z    +0.000, E1    -3.383, E3 +17727.822}
SPL {X  -159.990, Y  +384.811, Z    +0.000, E1   -11.531, E3 +17727.912}
SPL {X  -159.990, Y  +390.180, Z    +0.000, E1   -24.142, E3 +17728.216}
SPL {X  -159.990, Y  +397.074, Z    +0.000, E1   -39.012, E3 +17728.826}
SPL {X  -159.990, Y  +405.152, Z    +0.000, E1   -50.697, E3 +17729.965}
SPL {X  -159.990, Y  +423.293, Z    +0.000, E1   -63.280, E3 +17733.966}
SPL {X  -159.990, Y  +493.649, Z    +0.000, E1   -71.671, E3 +17759.670}
SPL {X  -159.990, Y  +662.531, Z    +0.000, E1   -73.010, E3 +17846.493}
SPL {X  -159.805, Y  +684.185, Z    +0.000, E1   -72.979, E3 +17860.777}
SPL {X  -158.739, Y  +696.464, Z    +0.000, E1   -72.862, E3 +17869.896}
SPL {X  -156.417, Y  +710.124, Z    +0.000, E1   -72.650, E3 +17881.119}
SPL {X  -153.206, Y  +722.596, Z    +0.000, E1   -72.287, E3 +17892.557}
SPL {X  -150.445, Y  +730.933, Z    +0.000, E1   -71.979, E3 +17900.768}
SPL {X  -147.389, Y  +738.737, Z    +0.000, E1   -71.634, E3 +17908.840}
SPL {X  -144.044, Y  +746.129, Z    +0.000, E1   -71.236, E3 +17916.835}
SPL {X  -140.684, Y  +752.689, Z    +0.000, E1   -70.820, E3 +17924.210}
SPL {X  -137.335, Y  +758.572, Z    +0.000, E1   -70.388, E3 +17931.017}
SPL {X  -134.566, Y  +763.037, Z    +0.000, E1   -70.007, E3 +17936.313}
SPL {X  -131.456, Y  +767.693, Z    +0.000, E1   -69.587, E3 +17941.877}
SPL {X  -127.440, Y  +773.226, Z    +0.000, E1   -69.006, E3 +17948.561}
SPL {X  -123.127, Y  +778.659, Z    +0.000, E1   -68.349, E3 +17955.103}
SPL {X   -80.879, Y  +814.541, Z    +0.000, E1   -55.704, E3 +18078.007}
ENDSPLINE

SPLINE
SPL {X  -125.518, Y  +775.707, Z    +0.000, E1   -52.189, E3 +18249.484}
SPL {X  -144.748, Y  +744.653, Z    +0.000, E1   -45.208, E3 +18267.680}
SPL {X  -153.147, Y  +722.791, Z    +0.000, E1   -36.417, E3 +18274.076}
SPL {X  -157.402, Y  +705.160, Z    +0.000, E1   -26.108, E3 +18277.171}
SPL {X  -159.480, Y  +689.270, Z    +0.000, E1   -14.023, E3 +18278.737}
SPL {X  -159.986, Y  +677.650, Z    +0.000, E1    -3.291, E3 +18279.231}
SPL {X  -159.990, Y  +674.500, Z    +0.000, E1    +0.000, E3 +18279.262}
SPL {X  -159.990, Y  +672.716, Z    +0.000, E1    +3.405, E3 +18279.278}
SPL {X  -159.990, Y  +668.521, Z    +0.000, E1   +13.007, E3 +18279.397}
SPL {X  -159.990, Y  +662.839, Z    +0.000, E1   +26.519, E3 +18279.740}
SPL {X  -159.990, Y  +653.836, Z    +0.000, E1   +43.967, E3 +18280.670}
SPL {X  -159.990, Y  +641.022, Z    +0.000, E1   +57.726, E3 +18282.979}
SPL {X  -159.990, Y  +617.987, Z    +0.000, E1   +67.134, E3 +18288.874}
SPL {X  -159.990, Y  +532.407, Z    +0.000, E1   +73.084, E3 +18319.781}
SPL {X  -159.990, Y  +382.957, Z    +0.000, E1   +73.647, E3 +18396.041}
SPL {X  -159.615, Y  +366.548, Z    +0.000, E1   +73.602, E3 +18406.683}
SPL {X  -157.928, Y  +351.899, Z    +0.000, E1   +73.451, E3 +18417.537}
ENDSPLINE

SPLINE
SPL {X  -159.990, Y  +380.170, Z    +0.000, E1   +69.785, E3 +18433.678}
ENDSPLINE

SPLINE
SPL {X  -158.227, Y  +353.814, Z    +0.000, E1   +70.663, E3 +18445.571}
SPL {X  -155.560, Y  +340.111, Z    +0.000, E1   +70.976, E3 +18452.593}
SPL {X  -151.918, Y  +327.322, Z    +0.000, E1   +71.266, E3 +18458.937}
SPL {X  -144.697, Y  +309.238, Z    +0.000, E1   +71.848, E3 +18465.886}
SPL {X  -140.298, Y  +300.601, Z    +0.000, E1   +71.461, E3 +18474.174}
SPL {X  -135.903, Y  +293.078, Z    +0.000, E1   +70.930, E3 +18482.712}
SPL {X  -130.487, Y  +284.926, Z    +0.000, E1   +70.202, E3 +18492.271}
SPL {X  -125.807, Y  +278.659, Z    +0.000, E1   +69.508, E3 +18499.727}
SPL {X  -122.967, Y  +275.148, Z    +0.000, E1   +69.053, E3 +18503.896}
SPL {X  -121.236, Y  +273.103, Z    +0.000, E1   +68.779, E3 +18506.282}
SPL {X   -84.117, Y  +241.407, Z    +0.000, E1   +58.224, E3 +18595.988}
ENDSPLINE

SPLINE
SPL {X  -106.708, Y  +258.294, Z    +0.000, E1   +53.789, E3 +18774.775}
SPL {X  -137.973, Y  +296.505, Z    +0.000, E1   +48.844, E3 +18813.555}
SPL {X  -150.692, Y  +323.752, Z    +0.000, E1   +39.895, E3 +18823.920}
SPL {X  -157.053, Y  +346.986, Z    +0.000, E1   +27.437, E3 +18828.400}
SPL {X  -159.518, Y  +365.226, Z    +0.000, E1   +13.562, E3 +18830.266}
SPL {X  -159.976, Y  +375.387, Z    +0.000, E1    +4.229, E3 +18830.701}
SPL {X  -159.990, Y  +379.485, Z    +0.000, E1    +0.028, E3 +18830.746}
SPL {X  -159.990, Y  +381.270, Z    +0.000, E1    -3.383, E3 +18830.764}
SPL {X  -159.990, Y  +384.811, Z    +0.000, E1   -11.531, E3 +18830.854}
SPL {X  -159.990, Y  +390.180, Z    +0.000, E1   -24.142, E3 +18831.157}
SPL {X  -159.990, Y  +397.074, Z    +0.000, E1   -39.012, E3 +18831.767}
SPL {X  -159.990, Y  +405.152, Z    +0.000, E1   -50.697, E3 +18832.906}
SPL {X  -159.990, Y  +423.293, Z    +0.000, E1   -63.280, E3 +18836.907}
SPL {X  -159.990, Y  +493.649, Z    +0.000, E1   -71.671, E3 +18862.611}
SPL {X  -159.990, Y  +662.531, Z    +0.000, E1   -73.010, E3 +18949.434}
SPL {X  -159.805, Y  +684.185, Z    +0.000, E1   -72.979, E3 +18963.718}
SPL {X  -158.295, Y  +699.729, Z    +0.000, E1   -72.830, E3 +18975.389}
SPL {X  -155.857, Y  +712.630, Z    +0.000, E1   -72.572, E3 +18986.318}
SPL {X  -153.206, Y  +722.596, Z    +0.000, E1   -72.287, E3 +18995.499}
SPL {X  -150.445, Y  +730.933, Z    +0.000, E1   -71.979, E3 +19003.709}
SPL {X  -147.389, Y  +738.737, Z    +0.000, E1   -71.634, E3 +19011.782}
SPL {X  -144.044, Y  +746.129, Z    +0.000, E1   -71.236, E3 +19019.776}
SPL {X  -140.684, Y  +752.689, Z    +0.000, E1   -70.820, E3 +19027.151}
SPL {X  -137.335, Y  +758.572, Z    +0.000, E1   -70.388, E3 +19033.959}
SPL {X  -133.651, Y  +764.444, Z    +0.000, E1   -69.897, E3 +19040.911}
SPL {X  -129.492, Y  +770.461, Z    +0.000, E1   -69.311, E3 +19048.151}
SPL {X  -125.168, Y  +776.148, Z    +0.000, E1   -68.666, E3 +19055.027}
SPL {X  -122.036, Y  +779.960, Z    +0.000, E1   -68.144, E3 +19059.631}
SPL {X   -80.879, Y  +814.541, Z    +0.000, E1   -55.704, E3 +19180.948}
ENDSPLINE

SPLINE
SPL {X  -125.518, Y  +775.707, Z    +0.000, E1   -52.189, E3 +19352.426}
SPL {X  -144.748, Y  +744.653, Z    +0.000, E1   -45.208, E3 +19370.621}
SPL {X  -153.147, Y  +722.791, Z    +0.000, E1   -36.417, E3 +19377.017}
SPL {X  -157.402, Y  +705.160, Z    +0.000, E1   -26.108, E3 +19380.112}
SPL {X  -159.480, Y  +689.270, Z    +0.000, E1   -14.023, E3 +19381.678}
SPL {X  -159.986, Y  +677.650, Z    +0.000, E1    -3.291, E3 +19382.172}
SPL {X  -159.990, Y  +674.500, Z    +0.000, E1    +0.000, E3 +19382.203}
SPL {X  -159.990, Y  +672.716, Z    +0.000, E1    +3.405, E3 +19382.219}
SPL {X  -159.990, Y  +668.521, Z    +0.000, E1   +13.007, E3 +19382.338}
SPL {X  -159.990, Y  +664.286, Z    +0.000, E1   +23.338, E3 +19382.570}
SPL {X  -159.990, Y  +658.431, Z    +0.000, E1   +35.998, E3 +19383.065}
SPL {X  -159.990, Y  +650.524, Z    +0.000, E1   +48.779, E3 +19384.053}
SPL {X  -159.990, Y  +641.022, Z    +0.000, E1   +57.726, E3 +19385.920}
SPL {X  -159.990, Y  +617.987, Z    +0.000, E1   +67.134, E3 +19391.815}
SPL {X  -159.990, Y  +532.407, Z    +0.000, E1   +73.084, E3 +19422.722}
SPL {X  -159.990, Y  +390.607, Z    +0.000, E1   +73.632, E3 +19494.258}
SPL {X  -159.886, Y  +371.742, Z    +0.000, E1   +73.650, E3 +19506.045}
SPL {X  -157.928, Y  +351.899, Z    +0.000, E1   +73.451, E3 +19520.479}
ENDSPLINE

SPLINE
SPL {X  -159.990, Y  +380.170, Z    +0.000, E1   +69.785, E3 +19536.619}
ENDSPLINE

SPLINE
SPL {X  -158.227, Y  +353.814, Z    +0.000, E1   +70.663, E3 +19548.512}
SPL {X  -155.560, Y  +340.111, Z    +0.000, E1   +70.976, E3 +19555.534}
SPL {X  -151.918, Y  +327.322, Z    +0.000, E1   +71.266, E3 +19561.878}
SPL {X  -144.697, Y  +309.238, Z    +0.000, E1   +71.848, E3 +19568.828}
SPL {X  -140.298, Y  +300.601, Z    +0.000, E1   +71.461, E3 +19577.115}
SPL {X  -135.903, Y  +293.078, Z    +0.000, E1   +70.930, E3 +19585.653}
SPL {X  -130.487, Y  +284.926, Z    +0.000, E1   +70.202, E3 +19595.212}
SPL {X  -125.807, Y  +278.659, Z    +0.000, E1   +69.508, E3 +19602.669}
SPL {X  -122.967, Y  +275.148, Z    +0.000, E1   +69.053, E3 +19606.837}
SPL {X  -121.236, Y  +273.103, Z    +0.000, E1   +68.779, E3 +19609.223}
SPL {X   -84.117, Y  +241.407, Z    +0.000, E1   +58.224, E3 +19698.929}
ENDSPLINE

SPLINE
SPL {X  -116.986, Y  +268.362, Z    +0.000, E1   +53.233, E3 +19892.844}
SPL {X  -146.319, Y  +312.789, Z    +0.000, E1   +44.152, E3 +19923.310}
SPL {X  -157.053, Y  +346.986, Z    +0.000, E1   +27.437, E3 +19931.342}
SPL {X  -159.518, Y  +365.226, Z    +0.000, E1   +13.562, E3 +19933.207}
SPL {X  -159.976, Y  +375.387, Z    +0.000, E1    +4.229, E3 +19933.643}
SPL {X  -159.990, Y  +379.485, Z    +0.000, E1    +0.028, E3 +19933.688}
SPL {X  -159.990, Y  +381.270, Z    +0.000, E1    -3.383, E3 +19933.705}
SPL {X  -159.990, Y  +384.811, Z    +0.000, E1   -11.531, E3 +19933.795}
SPL {X  -159.990, Y  +388.002, Z    +0.000, E1   -19.281, E3 +19933.945}
SPL {X  -159.990, Y  +394.075, Z    +0.000, E1   -32.836, E3 +19934.423}
SPL {X  -159.990, Y  +405.152, Z    +0.000, E1   -50.697, E3 +19935.847}
SPL {X  -159.990, Y  +423.293, Z    +0.000, E1   -63.280, E3 +19939.849}
SPL {X  -159.990, Y  +493.649, Z    +0.000, E1   -71.671, E3 +19965.552}
SPL {X  -159.990, Y  +662.531, Z    +0.000, E1   -73.010, E3 +20052.376}
SPL {X  -159.805, Y  +684.185, Z    +0.000, E1   -72.979, E3 +20066.660}
SPL {X  -158.295, Y  +699.729, Z    +0.000, E1   -72.830, E3 +20078.330}
SPL {X  -155.857, Y  +712.630, Z    +0.000, E1   -72.572, E3 +20089.259}
SPL {X  -153.206, Y  +722.596, Z    +0.000, E1   -72.287, E3 +20098.440}
SPL {X  -150.445, Y  +730.933, Z    +0.000, E1   -71.979, E3 +20106.650}
SPL {X  -147.389, Y  +738.737, Z    +0.000, E1   -71.634, E3 +20114.723}
SPL {X  -144.044, Y  +746.129, Z    +0.000, E1   -71.236, E3 +20122.717}
SPL {X  -140.684, Y  +752.689, Z    +0.000, E1   -70.820, E3 +20130.092}
SPL {X  -136.099, Y  +760.606, Z    +0.000, E1   -70.253, E3 +20139.248}
SPL {X  -131.456, Y  +767.693, Z    +0.000, E1   -69.587, E3 +20147.760}
SPL {X  -127.440, Y  +773.226, Z    +0.000, E1   -69.006, E3 +20154.443}
SPL {X  -123.127, Y  +778.659, Z    +0.000, E1   -68.349, E3 +20160.985}
SPL {X   -80.879, Y  +814.541, Z    +0.000, E1   -55.704, E3 +20283.889}
ENDSPLINE

SPLINE
SPL {X  -125.518, Y  +775.707, Z    +0.000, E1   -52.189, E3 +20455.367}
SPL {X  -144.748, Y  +744.653, Z    +0.000, E1   -45.208, E3 +20473.563}
SPL {X  -153.147, Y  +722.791, Z    +0.000, E1   -36.417, E3 +20479.958}
SPL {X  -158.456, Y  +698.602, Z    +0.000, E1   -21.523, E3 +20483.804}
SPL {X  -159.738, Y  +685.469, Z    +0.000, E1   -10.595, E3 +20484.859}
SPL {X  -159.986, Y  +677.650, Z    +0.000, E1    -3.291, E3 +20485.114}
SPL {X  -159.990, Y  +674.500, Z    +0.000, E1    +0.000, E3 +20485.144}
SPL {X  -159.990, Y  +672.716, Z    +0.000, E1    +3.405, E3 +20485.161}
SPL {X  -159.990, Y  +668.521, Z    +0.000, E1   +13.007, E3 +20485.280}
SPL {X  -159.990, Y  +664.286, Z    +0.000, E1   +23.338, E3 +20485.511}
SPL {X  -159.990, Y  +658.431, Z    +0.000, E1   +35.998, E3 +20486.006}
SPL {X  -159.990, Y  +650.524, Z    +0.000, E1   +48.779, E3 +20486.994}
SPL {X  -159.990, Y  +641.022, Z    +0.000, E1   +57.726, E3 +20488.861}
SPL {X  -159.990, Y  +617.987, Z    +0.000, E1   +67.134, E3 +20494.757}
SPL {X  -159.990, Y  +532.407, Z    +0.000, E1   +73.084, E3 +20525.663}
SPL {X  -159.990, Y  +390.607, Z    +0.000, E1   +73.632, E3 +20597.199}
SPL {X  -159.886, Y  +371.742, Z    +0.000, E1   +73.650, E3 +20608.986}
SPL {X  -157.928, Y  +351.899, Z    +0.000, E1   +73.451, E3 +20623.420}
ENDSPLINE

SPLINE
SPL {X  -159.990, Y  +380.170, Z    +0.000, E1   +69.785, E3 +20639.560}
ENDSPLINE

SPLINE
SPL {X  -158.227, Y  +353.814, Z    +0.000, E1   +70.663, E3 +20651.454}
SPL {X  -154.257, Y  +335.055, Z    +0.000, E1   +71.089, E3 +20661.082}
SPL {X  -148.153, Y  +317.104, Z    +0.000, E1   +71.658, E3 +20668.227}
SPL {X  -143.479, Y  +306.716, Z    +0.000, E1   +71.847, E3 +20673.301}
SPL {X  -140.298, Y  +300.601, Z    +0.000, E1   +71.461, E3 +20680.056}
SPL {X  -137.001, Y  +294.872, Z    +0.000, E1   +71.048, E3 +20686.564}
SPL {X  -133.301, Y  +289.026, Z    +0.000, E1   +70.567, E3 +20693.351}
SPL {X  -128.648, Y  +282.387, Z    +0.000, E1   +69.939, E3 +20701.166}
SPL {X  -125.063, Y  +277.720, Z    +0.000, E1   +69.378, E3 +20706.742}
SPL {X  -122.086, Y  +274.099, Z    +0.000, E1   +68.932, E3 +20710.987}
SPL {X   -84.117, Y  +241.407, Z    +0.000, E1   +58.224, E3 +20801.870}
ENDSPLINE

SPLINE
SPL {X  -106.708, Y  +258.294, Z    +0.000, E1   +53.789, E3 +20980.657}
SPL {X  -137.973, Y  +296.505, Z    +0.000, E1   +48.844, E3 +21019.437}
SPL {X  -154.359, Y  +335.426, Z    +0.000, E1   +34.338, E3 +21032.333}
SPL {X  -159.279, Y  +362.429, Z    +0.000, E1   +16.013, E3 +21035.933}
SPL {X  -159.976, Y  +375.387, Z    +0.000, E1    +4.229, E3 +21036.584}
SPL {X  -159.990, Y  +379.485, Z    +0.000, E1    +0.028, E3 +21036.629}
SPL {X  -159.990, Y  +381.270, Z    +0.000, E1    -3.383, E3 +21036.646}
SPL {X  -159.990, Y  +386.246, Z    +0.000, E1   -14.704, E3 +21036.803}
SPL {X  -159.990, Y  +394.075, Z    +0.000, E1   -32.836, E3 +21037.364}
SPL {X  -159.990, Y  +405.152, Z    +0.000, E1   -50.697, E3 +21038.788}
SPL {X  -159.990, Y  +423.293, Z    +0.000, E1   -63.280, E3 +21042.790}
SPL {X  -159.990, Y  +493.649, Z    +0.000, E1   -71.671, E3 +21068.494}
SPL {X  -159.990, Y  +662.531, Z    +0.000, E1   -73.010, E3 +21155.317}
SPL {X  -159.805, Y  +684.185, Z    +0.000, E1   -72.979, E3 +21169.601}
SPL {X  -158.739, Y  +696.464, Z    +0.000, E1   -72.862, E3 +21178.719}
SPL {X  -156.417, Y  +710.124, Z    +0.000, E1   -72.650, E3 +21189.943}
SPL {X  -153.206, Y  +722.596, Z    +0.000, E1   -72.287, E3 +21201.381}
SPL {X  -150.445, Y  +730.933, Z    +0.000, E1   -71.979, E3 +21209.591}
SPL {X  -147.389, Y  +738.737, Z    +0.000, E1   -71.634, E3 +21217.664}
SPL {X  -144.044, Y  +746.129, Z    +0.000, E1   -71.236, E3 +21225.658}
SPL {X  -140.684, Y  +752.689, Z    +0.000, E1   -70.820, E3 +21233.034}
SPL {X  -137.335, Y  +758.572, Z    +0.000, E1   -70.388, E3 +21239.841}
SPL {X  -133.651, Y  +764.444, Z    +0.000, E1   -69.897, E3 +21246.793}
SPL {X  -130.650, Y  +768.844, Z    +0.000, E1   -69.455, E3 +21252.114}
SPL {X  -127.440, Y  +773.226, Z    +0.000, E1   -69.006, E3 +21257.385}
SPL {X  -123.127, Y  +778.659, Z    +0.000, E1   -68.349, E3 +21263.927}
SPL {X   -80.879, Y  +814.541, Z    +0.000, E1   -55.704, E3 +21386.831}
ENDSPLINE

SPLINE
SPL {X  -125.518, Y  +775.707, Z    +0.000, E1   -52.189, E3 +21558.308}
SPL {X  -150.797, Y  +729.951, Z    +0.000, E1   -39.777, E3 +21581.043}
SPL {X  -158.456, Y  +698.602, Z    +0.000, E1   -21.523, E3 +21586.746}
SPL {X  -159.738, Y  +685.469, Z    +0.000, E1   -10.595, E3 +21587.800}
SPL {X  -159.986, Y  +677.650, Z    +0.000, E1    -3.291, E3 +21588.055}
SPL {X  -159.990, Y  +674.500, Z    +0.000, E1    +0.000, E3 +21588.085}
SPL {X  -159.990, Y  +672.716, Z    +0.000, E1    +3.405, E3 +21588.102}
SPL {X  -159.990, Y  +668.521, Z    +0.000, E1   +13.007, E3 +21588.221}
SPL {X  -159.990, Y  +662.839, Z    +0.000, E1   +26.519, E3 +21588.563}
SPL {X  -159.990, Y  +653.836, Z    +0.000, E1   +43.967, E3 +21589.493}
SPL {X  -159.990, Y  +641.022, Z    +0.000, E1   +57.726, E3 +21591.802}
SPL {X  -159.990, Y  +617.987, Z    +0.000, E1   +67.134, E3 +21597.698}
SPL {X  -159.990, Y  +532.407, Z    +0.000, E1   +73.084, E3 +21628.605}
SPL {X  -159.990, Y  +382.957, Z    +0.000, E1   +73.647, E3 +21704.864}
SPL {X  -159.615, Y  +366.548, Z    +0.000, E1   +73.602, E3 +21715.507}
SPL {X  -157.928, Y  +351.899, Z    +0.000, E1   +73.451, E3 +21726.361}
ENDSPLINE

SPLINE
SPL {X  -159.990, Y  +380.170, Z    +0.000, E1   +69.785, E3 +21742.501}
ENDSPLINE

SPLINE
SPL {X  -158.227, Y  +353.814, Z    +0.000, E1   +70.663, E3 +21754.395}
SPL {X  -154.257, Y  +335.055, Z    +0.000, E1   +71.089, E3 +21764.023}
SPL {X  -148.153, Y  +317.104, Z    +0.000, E1   +71.658, E3 +21771.168}
SPL {X  -143.479, Y  +306.716, Z    +0.000, E1   +71.847, E3 +21776.242}
SPL {X  -140.298, Y  +300.601, Z    +0.000, E1   +71.461, E3 +21782.997}
SPL {X  -137.001, Y  +294.872, Z    +0.000, E1   +71.048, E3 +21789.506}
SPL {X  -133.301, Y  +289.026, Z    +0.000, E1   +70.567, E3 +21796.292}
SPL {X  -129.603, Y  +283.692, Z    +0.000, E1   +70.051, E3 +21802.592}
SPL {X  -125.807, Y  +278.659, Z    +0.000, E1   +69.508, E3 +21808.551}
SPL {X  -122.086, Y  +274.099, Z    +0.000, E1   +68.932, E3 +21813.928}
SPL {X   -84.117, Y  +241.407, Z    +0.000, E1   +58.224, E3 +21904.811}
ENDSPLINE

SPLINE
SPL {X  -116.986, Y  +268.362, Z    +0.000, E1   +53.233, E3 +22098.727}
SPL {X  -146.319, Y  +312.789, Z    +0.000, E1   +44.152, E3 +22129.193}
SPL {X  -157.053, Y  +346.986, Z    +0.000, E1   +27.437, E3 +22137.224}
SPL {X  -159.518, Y  +365.226, Z    +0.000, E1   +13.562, E3 +22139.089}
SPL {X  -159.976, Y  +375.387, Z    +0.000, E1    +4.229, E3 +22139.525}
SPL {X  -159.990, Y  +379.485, Z    +0.000, E1    +0.028, E3 +22139.570}
SPL {X  -159.990, Y  +381.270, Z    +0.000, E1    -3.383, E3 +22139.587}
SPL {X  -159.990, Y  +386.246, Z    +0.000, E1   -14.704, E3 +22139.745}
SPL {X  -159.990, Y  +394.075, Z    +0.000, E1   -32.836, E3 +22140.305}
SPL {X  -159.990, Y  +405.152, Z    +0.000, E1   -50.697, E3 +22141.730}
SPL {X  -159.990, Y  +423.293, Z    +0.000, E1   -63.280, E3 +22145.731}
SPL {X  -159.990, Y  +493.649, Z    +0.000, E1   -71.671, E3 +22171.435}
SPL {X  -159.990, Y  +662.531, Z    +0.000, E1   -73.010, E3 +22258.258}
SPL {X  -159.805, Y  +684.185, Z    +0.000, E1   -72.979, E3 +22272.542}
SPL {X  -158.295, Y  +699.729, Z    +0.000, E1   -72.830, E3 +22284.212}
SPL {X  -155.857, Y  +712.630, Z    +0.000, E1   -72.572, E3 +22295.141}
SPL {X  -153.206, Y  +722.596, Z    +0.000, E1   -72.287, E3 +22304.322}
SPL {X  -150.445, Y  +730.933, Z    +0.000, E1   -71.979, E3 +22312.532}
SPL {X  -147.389, Y  +738.737, Z    +0.000, E1   -71.634, E3 +22320.605}
SPL {X  -144.044, Y  +746.129, Z    +0.000, E1   -71.236, E3 +22328.600}
SPL {X  -140.684, Y  +752.689, Z    +0.000, E1   -70.820, E3 +22335.975}
SPL {X  -137.335, Y  +758.572, Z    +0.000, E1   -70.388, E3 +22342.782}
SPL {X  -134.566, Y  +763.037, Z    +0.000, E1   -70.007, E3 +22348.078}
SPL {X  -131.456, Y  +767.693, Z    +0.000, E1   -69.587, E3 +22353.642}
SPL {X  -127.440, Y  +773.226, Z    +0.000, E1   -69.006, E3 +22360.326}
SPL {X  -123.127, Y  +778.659, Z    +0.000, E1   -68.349, E3 +22366.868}
SPL {X   -80.879, Y  +814.541, Z    +0.000, E1   -55.704, E3 +22489.772}
ENDSPLINE

SPLINE
SPL {X  -125.518, Y  +775.707, Z    +0.000, E1   -52.189, E3 +22661.249}
SPL {X  -150.797, Y  +729.951, Z    +0.000, E1   -39.777, E3 +22683.984}
SPL {X  -158.456, Y  +698.602, Z    +0.000, E1   -21.523, E3 +22689.687}
SPL {X  -159.738, Y  +685.469, Z    +0.000, E1   -10.595, E3 +22690.741}
SPL {X  -159.986, Y  +677.650, Z    +0.000, E1    -3.291, E3 +22690.996}
SPL {X  -159.990, Y  +674.500, Z    +0.000, E1    +0.000, E3 +22691.026}
SPL {X  -159.990, Y  +672.716, Z    +0.000, E1    +3.405, E3 +22691.043}
SPL {X  -159.990, Y  +668.521, Z    +0.000, E1   +13.007, E3 +22691.162}
SPL {X  -159.990, Y  +664.286, Z    +0.000, E1   +23.338, E3 +22691.393}
SPL {X  -159.990, Y  +658.431, Z    +0.000, E1   +35.998, E3 +22691.888}
SPL {X  -159.990, Y  +650.524, Z    +0.000, E1   +48.779, E3 +22692.877}
SPL {X  -159.990, Y  +641.022, Z    +0.000, E1   +57.726, E3 +22694.743}
SPL {X  -159.990, Y  +617.987, Z    +0.000, E1   +67.134, E3 +22700.639}
SPL {X  -159.990, Y  +532.407, Z    +0.000, E1   +73.084, E3 +22731.546}
SPL {X  -159.990, Y  +390.607, Z    +0.000, E1   +73.632, E3 +22803.082}
SPL {X  -159.886, Y  +371.742, Z    +0.000, E1   +73.650, E3 +22814.869}
SPL {X  -157.928, Y  +351.899, Z    +0.000, E1   +73.451, E3 +22829.302}
ENDSPLINE

SPLINE
SPL {X  -159.990, Y  +387.996, Z    +0.000, E1   +69.509, E3 +22841.732}
ENDSPLINE

SPLINE
SPL {X  -159.889, Y  +371.819, Z    +0.000, E1   +70.046, E3 +22849.459}
SPL {X  -158.227, Y  +353.814, Z    +0.000, E1   +70.663, E3 +22857.336}
SPL {X  -155.560, Y  +340.111, Z    +0.000, E1   +70.976, E3 +22864.358}
SPL {X  -151.918, Y  +327.322, Z    +0.000, E1   +71.266, E3 +22870.702}
SPL {X  -144.697, Y  +309.238, Z    +0.000, E1   +71.848, E3 +22877.651}
SPL {X  -140.298, Y  +300.601, Z    +0.000, E1   +71.461, E3 +22885.939}
SPL {X  -135.903, Y  +293.078, Z    +0.000, E1   +70.930, E3 +22894.476}
SPL {X  -130.487, Y  +284.926, Z    +0.000, E1   +70.202, E3 +22904.036}
SPL {X  -125.807, Y  +278.659, Z    +0.000, E1   +69.508, E3 +22911.492}
SPL {X  -122.086, Y  +274.099, Z    +0.000, E1   +68.932, E3 +22916.870}
SPL {X   -84.117, Y  +241.407, Z    +0.000, E1   +58.224, E3 +23007.752}
ENDSPLINE

SPLINE
SPL {X  -106.708, Y  +258.294, Z    +0.000, E1   +53.789, E3 +23186.539}
SPL {X  -137.973, Y  +296.505, Z    +0.000, E1   +48.844, E3 +23225.319}
SPL {X  -154.359, Y  +335.426, Z    +0.000, E1   +34.338, E3 +23238.215}
SPL {X  -159.279, Y  +362.429, Z    +0.000, E1   +16.013, E3 +23241.815}
SPL {X  -159.976, Y  +375.387, Z    +0.000, E1    +4.229, E3 +23242.466}
SPL {X  -159.990, Y  +379.485, Z    +0.000, E1    +0.028, E3 +23242.511}
SPL {X  -159.990, Y  +381.270, Z    +0.000, E1    -3.383, E3 +23242.528}
SPL {X  -159.990, Y  +386.246, Z    +0.000, E1   -14.704, E3 +23242.686}
SPL {X  -159.990, Y  +394.075, Z    +0.000, E1   -32.836, E3 +23243.246}
SPL {X  -159.990, Y  +405.152, Z    +0.000, E1   -50.697, E3 +23244.671}
SPL {X  -159.990, Y  +423.293, Z    +0.000, E1   -63.280, E3 +23248.672}
SPL {X  -159.990, Y  +493.649, Z    +0.000, E1   -71.671, E3 +23274.376}
SPL {X  -159.990, Y  +662.531, Z    +0.000, E1   -73.010, E3 +23361.199}
SPL {X  -159.805, Y  +684.185, Z    +0.000, E1   -72.979, E3 +23375.483}
SPL {X  -158.295, Y  +699.729, Z    +0.000, E1   -72.830, E3 +23387.153}
SPL {X  -155.857, Y  +712.630, Z    +0.000, E1   -72.572, E3 +23398.082}
SPL {X  -153.206, Y  +722.596, Z    +0.000, E1   -72.287, E3 +23407.263}
SPL {X  -150.445, Y  +730.933, Z    +0.000, E1   -71.979, E3 +23415.474}
SPL {X  -147.389, Y  +738.737, Z    +0.000, E1   -71.634, E3 +23423.546}
SPL {X  -144.044, Y  +746.129, Z    +0.000, E1   -71.236, E3 +23431.541}
SPL {X  -140.684, Y  +752.689, Z    +0.000, E1   -70.820, E3 +23438.916}
SPL {X  -136.099, Y  +760.606, Z    +0.000, E1   -70.253, E3 +23448.071}
SPL {X  -131.456, Y  +767.693, Z    +0.000, E1   -69.587, E3 +23456.583}
SPL {X  -128.507, Y  +771.803, Z    +0.000, E1   -69.145, E3 +23461.565}
SPL {X  -125.168, Y  +776.148, Z    +0.000, E1   -68.666, E3 +23466.792}
SPL {X  -122.036, Y  +779.960, Z    +0.000, E1   -68.144, E3 +23471.395}
SPL {X   -80.879, Y  +814.541, Z    +0.000, E1   -55.704, E3 +23592.713}
ENDSPLINE

SPLINE
SPL {X  -125.518, Y  +775.707, Z    +0.000, E1   -52.189, E3 +23764.190}
SPL {X  -150.797, Y  +729.951, Z    +0.000, E1   -39.777, E3 +23786.925}
SPL {X  -158.456, Y  +698.602, Z    +0.000, E1   -21.523, E3 +23792.628}
SPL {X  -159.738, Y  +685.469, Z    +0.000, E1   -10.595, E3 +23793.682}
SPL {X  -159.986, Y  +677.650, Z    +0.000, E1    -3.291, E3 +23793.937}
SPL {X  -159.990, Y  +674.500, Z    +0.000, E1    +0.000, E3 +23793.968}
SPL {X  -159.990, Y  +672.716, Z    +0.000, E1    +3.405, E3 +23793.984}
SPL {X  -159.990, Y  +668.521, Z    +0.000, E1   +13.007, E3 +23794.103}
SPL {X  -159.990, Y  +662.839, Z    +0.000, E1   +26.519, E3 +23794.445}
SPL {X  -159.990, Y  +653.836, Z    +0.000, E1   +43.967, E3 +23795.376}
SPL {X  -159.990, Y  +641.022, Z    +0.000, E1   +57.726, E3 +23797.685}
SPL {X  -159.990, Y  +617.987, Z    +0.000, E1   +67.134, E3 +23803.580}
SPL {X  -159.990, Y  +532.407, Z    +0.000, E1   +73.084, E3 +23834.487}
SPL {X  -159.990, Y  +390.607, Z    +0.000, E1   +73.632, E3 +23906.023}
SPL {X  -159.886, Y  +371.742, Z    +0.000, E1   +73.650, E3 +23917.810}
SPL {X  -157.928, Y  +351.899, Z    +0.000, E1   +73.451, E3 +23932.243}
ENDSPLINE

SPLINE
SPL {X  -159.990, Y  +387.996, Z    +0.000, E1   +69.509, E3 +23944.673}
ENDSPLINE

SPLINE
SPL {X  -159.889, Y  +371.819, Z    +0.000, E1   +70.046, E3 +23952.400}
SPL {X  -158.227, Y  +353.814, Z    +0.000, E1   +70.663, E3 +23960.277}
SPL {X  -154.257, Y  +335.055, Z    +0.000, E1   +71.089, E3 +23969.905}
SPL {X  -148.153, Y  +317.104, Z    +0.000, E1   +71.658, E3 +23977.051}
SPL {X  -143.479, Y  +306.716, Z    +0.000, E1   +71.847, E3 +23982.124}
SPL {X  -140.298, Y  +300.601, Z    +0.000, E1   +71.461, E3 +23988.880}
SPL {X  -135.903, Y  +293.078, Z    +0.000, E1   +70.930, E3 +23997.417}
SPL {X  -130.487, Y  +284.926, Z    +0.000, E1   +70.202, E3 +24006.977}
SPL {X  -125.807, Y  +278.659, Z    +0.000, E1   +69.508, E3 +24014.433}
SPL {X  -122.086, Y  +274.099, Z    +0.000, E1   +68.932, E3 +24019.811}
SPL {X   -84.117, Y  +241.407, Z    +0.000, E1   +58.224, E3 +24110.693}
ENDSPLINE

SPLINE
SPL {X  -106.708, Y  +258.294, Z    +0.000, E1   +53.789, E3 +24289.480}
SPL {X  -137.973, Y  +296.505, Z    +0.000, E1   +48.844, E3 +24328.261}
SPL {X  -150.692, Y  +323.752, Z    +0.000, E1   +39.895, E3 +24338.626}
SPL {X  -157.053, Y  +346.986, Z    +0.000, E1   +27.437, E3 +24343.106}
SPL {X  -159.518, Y  +365.226, Z    +0.000, E1   +13.562, E3 +24344.972}
SPL {X  -159.976, Y  +375.387, Z    +0.000, E1    +4.229, E3 +24345.407}
SPL {X  -159.990, Y  +379.485, Z    +0.000, E1    +0.028, E3 +24345.452}
SPL {X  -159.990, Y  +381.270, Z    +0.000, E1    -3.383, E3 +24345.469}
SPL {X  -159.990, Y  +384.811, Z    +0.000, E1   -11.531, E3 +24345.560}
SPL {X  -159.990, Y  +390.180, Z    +0.000, E1   -24.142, E3 +24345.863}
SPL {X  -159.990, Y  +397.074, Z    +0.000, E1   -39.012, E3 +24346.473}
SPL {X  -159.990, Y  +405.152, Z    +0.000, E1   -50.697, E3 +24347.612}
SPL {X  -159.990, Y  +423.293, Z    +0.000, E1   -63.280, E3 +24351.613}
SPL {X  -159.990, Y  +493.649, Z    +0.000, E1   -71.671, E3 +24377.317}
SPL {X  -159.990, Y  +662.531, Z    +0.000, E1   -73.010, E3 +24464.140}
SPL {X  -159.805, Y  +684.185, Z    +0.000, E1   -72.979, E3 +24478.424}
SPL {X  -158.295, Y  +699.729, Z    +0.000, E1   -72.830, E3 +24490.095}
SPL {X  -155.857, Y  +712.630, Z    +0.000, E1   -72.572, E3 +24501.024}
SPL {X  -153.206, Y  +722.596, Z    +0.000, E1   -72.287, E3 +24510.204}
SPL {X  -150.445, Y  +730.933, Z    +0.000, E1   -71.979, E3 +24518.415}
SPL {X  -147.389, Y  +738.737, Z    +0.000, E1   -71.634, E3 +24526.487}
SPL {X  -144.044, Y  +746.129, Z    +0.000, E1   -71.236, E3 +24534.482}
SPL {X  -140.684, Y  +752.689, Z    +0.000, E1   -70.820, E3 +24541.857}
SPL {X  -136.099, Y  +760.606, Z    +0.000, E1   -70.253, E3 +24551.013}
SPL {X  -131.456, Y  +767.693, Z    +0.000, E1   -69.587, E3 +24559.524}
SPL {X  -128.507, Y  +771.803, Z    +0.000, E1   -69.145, E3 +24564.506}
SPL {X  -125.168, Y  +776.148, Z    +0.000, E1   -68.666, E3 +24569.733}
SPL {X  -122.036, Y  +779.960, Z    +0.000, E1   -68.144, E3 +24574.336}
SPL {X   -80.879, Y  +814.541, Z    +0.000, E1   -55.704, E3 +24695.654}
ENDSPLINE

SPLINE
SPL {X  -125.518, Y  +775.707, Z    +0.000, E1   -52.189, E3 +24867.132}
SPL {X  -150.797, Y  +729.951, Z    +0.000, E1   -39.777, E3 +24889.866}
SPL {X  -158.456, Y  +698.602, Z    +0.000, E1   -21.523, E3 +24895.569}
SPL {X  -159.738, Y  +685.469, Z    +0.000, E1   -10.595, E3 +24896.623}
SPL {X  -159.986, Y  +677.650, Z    +0.000, E1    -3.291, E3 +24896.878}
SPL {X  -159.990, Y  +674.500, Z    +0.000, E1    +0.000, E3 +24896.909}
SPL {X  -159.990, Y  +672.716, Z    +0.000, E1    +3.405, E3 +24896.925}
SPL {X  -159.990, Y  +668.521, Z    +0.000, E1   +13.007, E3 +24897.044}
SPL {X  -159.990, Y  +662.839, Z    +0.000, E1   +26.519, E3 +24897.387}
SPL {X  -159.990, Y  +653.836, Z    +0.000, E1   +43.967, E3 +24898.317}
SPL {X  -159.990, Y  +641.022, Z    +0.000, E1   +57.726, E3 +24900.626}
SPL {X  -159.990, Y  +617.987, Z    +0.000, E1   +67.134, E3 +24906.521}
SPL {X  -159.990, Y  +532.407, Z    +0.000, E1   +73.084, E3 +24937.428}
SPL {X  -159.990, Y  +382.957, Z    +0.000, E1   +73.647, E3 +25013.688}
SPL {X  -159.615, Y  +366.548, Z    +0.000, E1   +73.602, E3 +25024.330}
SPL {X  -157.928, Y  +351.899, Z    +0.000, E1   +73.451, E3 +25035.184}
ENDSPLINE

SPLINE
SPL {X  -159.990, Y  +380.170, Z    +0.000, E1   +69.785, E3 +25051.325}
ENDSPLINE

SPLINE
SPL {X  -158.227, Y  +353.814, Z    +0.000, E1   +70.663, E3 +25063.218}
SPL {X  -154.257, Y  +335.055, Z    +0.000, E1   +71.089, E3 +25072.846}
SPL {X  -148.153, Y  +317.104, Z    +0.000, E1   +71.658, E3 +25079.992}
SPL {X  -143.479, Y  +306.716, Z    +0.000, E1   +71.847, E3 +25085.065}
SPL {X  -140.298, Y  +300.601, Z    +0.000, E1   +71.461, E3 +25091.821}
SPL {X  -137.001, Y  +294.872, Z    +0.000, E1   +71.048, E3 +25098.329}
SPL {X  -133.301, Y  +289.026, Z    +0.000, E1   +70.567, E3 +25105.116}
SPL {X  -128.648, Y  +282.387, Z    +0.000, E1   +69.939, E3 +25112.931}
SPL {X  -125.063, Y  +277.720, Z    +0.000, E1   +69.378, E3 +25118.507}
SPL {X  -122.086, Y  +274.099, Z    +0.000, E1   +68.932, E3 +25122.752}
SPL {X   -84.117, Y  +241.407, Z    +0.000, E1   +58.224, E3 +25213.635}
ENDSPLINE

